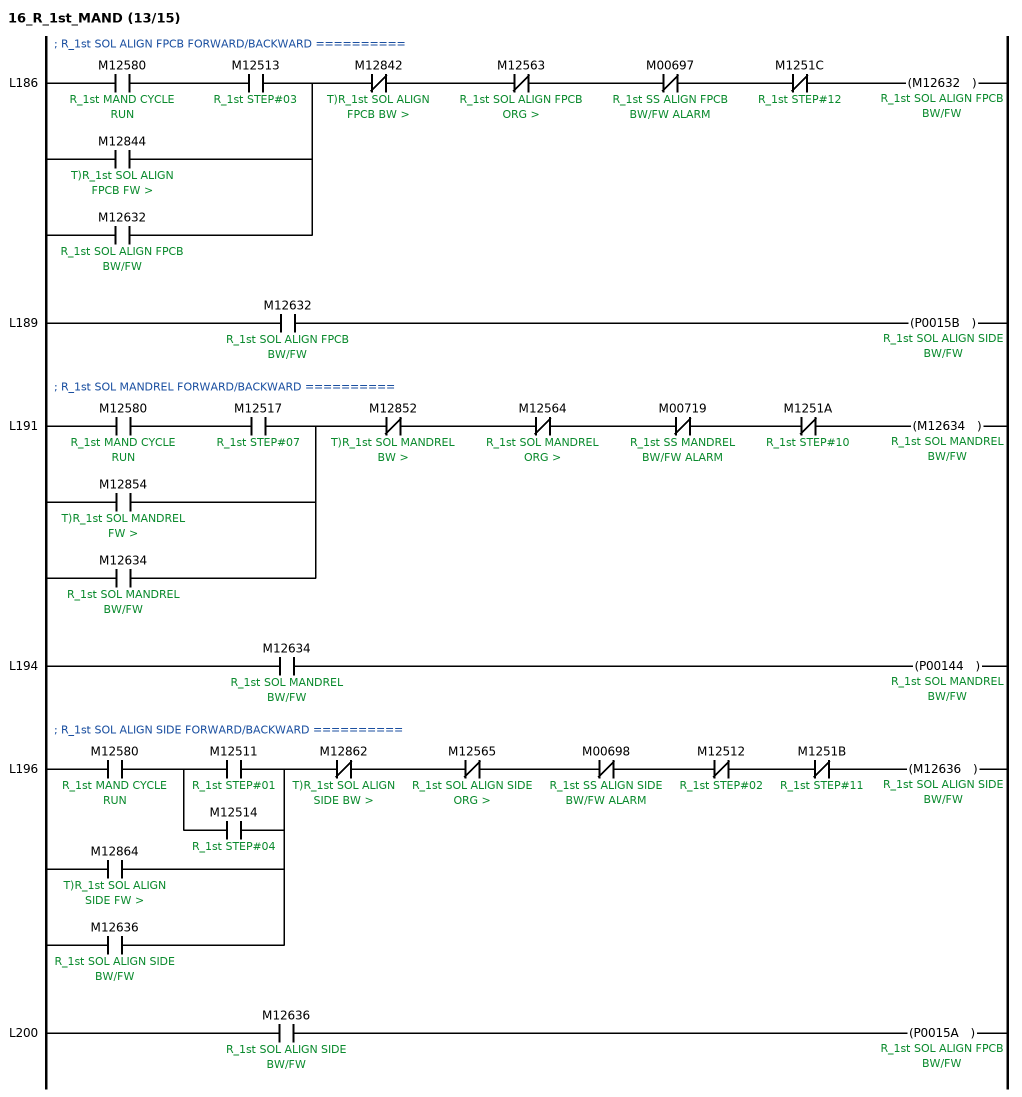
[picture p144: 16_R_1st_MAND rungs L186-L200]
// R_1st SOL ALIGN FPCB FORWARD/BACKWARD ==========
; L186
LOAD      M12580	// R_1st MAND CYCLE RUN
AND       M12513	// R_1st STEP#03
OR        M12844	// T)R_1st SOL ALIGN FPCB FW >
OR        M12632	// R_1st SOL ALIGN FPCB BW/FW
AND NOT   M12842	// T)R_1st SOL ALIGN FPCB BW >
AND NOT   M12563	// R_1st SOL ALIGN FPCB ORG >
AND NOT   M00697	// R_1st SS ALIGN FPCB BW/FW ALARM
AND NOT   M1251C	// R_1st STEP#12
OUT       M12632	// R_1st SOL ALIGN FPCB BW/FW
; L189
LOAD      M12632	// R_1st SOL ALIGN FPCB BW/FW
OUT       P0015B	// R_1st SOL ALIGN SIDE BW/FW
// R_1st SOL MANDREL FORWARD/BACKWARD ==========
; L191
LOAD      M12580	// R_1st MAND CYCLE RUN
AND       M12517	// R_1st STEP#07
OR        M12854	// T)R_1st SOL MANDREL FW >
OR        M12634	// R_1st SOL MANDREL BW/FW
AND NOT   M12852	// T)R_1st SOL MANDREL BW >
AND NOT   M12564	// R_1st SOL MANDREL ORG >
AND NOT   M00719	// R_1st SS MANDREL BW/FW ALARM
AND NOT   M1251A	// R_1st STEP#10
OUT       M12634	// R_1st SOL MANDREL BW/FW
; L194
LOAD      M12634	// R_1st SOL MANDREL BW/FW
OUT       P00144	// R_1st SOL MANDREL BW/FW
// R_1st SOL ALIGN SIDE FORWARD/BACKWARD ==========
; L196
LOAD      M12580	// R_1st MAND CYCLE RUN
LOAD      M12511	// R_1st STEP#01
OR        M12514	// R_1st STEP#04
AND LOAD
OR        M12864	// T)R_1st SOL ALIGN SIDE FW >
OR        M12636	// R_1st SOL ALIGN SIDE BW/FW
AND NOT   M12862	// T)R_1st SOL ALIGN SIDE BW >
AND NOT   M12565	// R_1st SOL ALIGN SIDE ORG >
AND NOT   M00698	// R_1st SS ALIGN SIDE BW/FW ALARM
AND NOT   M12512	// R_1st STEP#02
AND NOT   M1251B	// R_1st STEP#11
OUT       M12636	// R_1st SOL ALIGN SIDE BW/FW
; L200
LOAD      M12636	// R_1st SOL ALIGN SIDE BW/FW
OUT       P0015A	// R_1st SOL ALIGN FPCB BW/FW

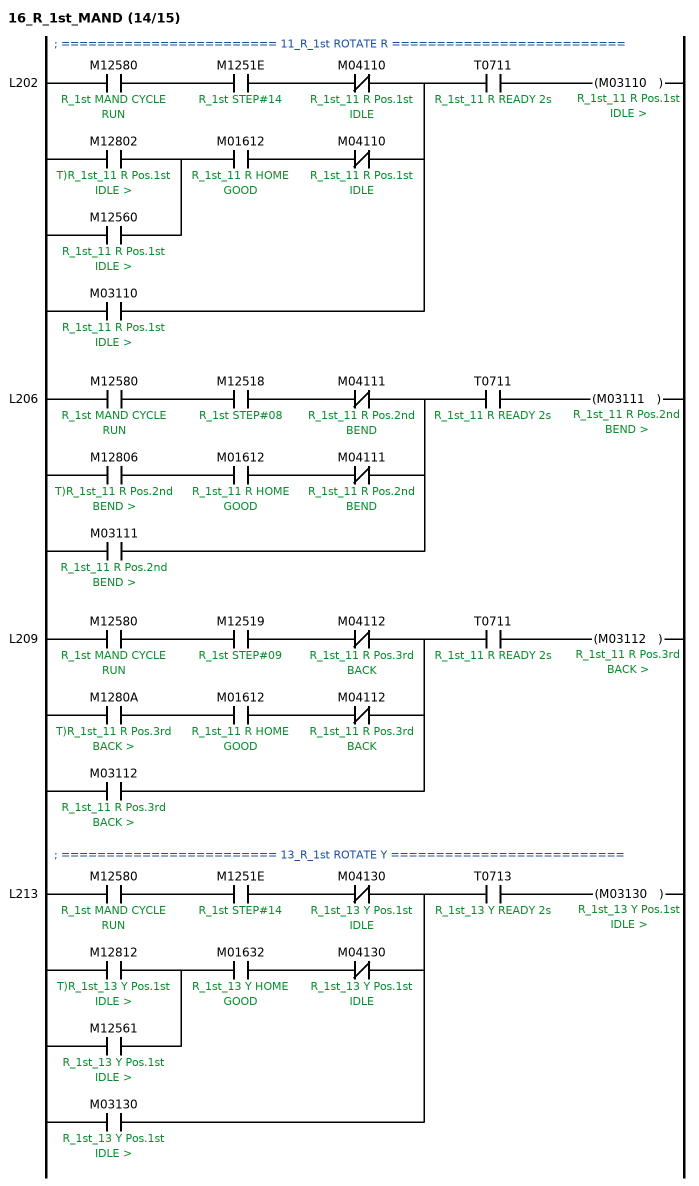
// ======================== 11_R_1st ROTATE R ==========================
; L202
LOAD      M12580	// R_1st MAND CYCLE RUN
AND       M1251E	// R_1st STEP#14
AND NOT   M04110	// R_1st_11 R Pos.1st IDLE
LOAD      M12802	// T)R_1st_11 R Pos.1st IDLE >
OR        M12560	// R_1st_11 R Pos.1st IDLE >
AND       M01612	// R_1st_11 R HOME GOOD
AND NOT   M04110	// R_1st_11 R Pos.1st IDLE
OR LOAD
OR        M03110	// R_1st_11 R Pos.1st IDLE >
AND       T0711	// R_1st_11 R READY 2s
OUT       M03110	// R_1st_11 R Pos.1st IDLE >
; L206
LOAD      M12580	// R_1st MAND CYCLE RUN
AND       M12518	// R_1st STEP#08
AND NOT   M04111	// R_1st_11 R Pos.2nd BEND
LOAD      M12806	// T)R_1st_11 R Pos.2nd BEND >
AND       M01612	// R_1st_11 R HOME GOOD
AND NOT   M04111	// R_1st_11 R Pos.2nd BEND
OR LOAD
OR        M03111	// R_1st_11 R Pos.2nd BEND >
AND       T0711	// R_1st_11 R READY 2s
OUT       M03111	// R_1st_11 R Pos.2nd BEND >
; L209
LOAD      M12580	// R_1st MAND CYCLE RUN
AND       M12519	// R_1st STEP#09
AND NOT   M04112	// R_1st_11 R Pos.3rd BACK
LOAD      M1280A	// T)R_1st_11 R Pos.3rd BACK >
AND       M01612	// R_1st_11 R HOME GOOD
AND NOT   M04112	// R_1st_11 R Pos.3rd BACK
OR LOAD
OR        M03112	// R_1st_11 R Pos.3rd BACK >
AND       T0711	// R_1st_11 R READY 2s
OUT       M03112	// R_1st_11 R Pos.3rd BACK >
// ======================== 13_R_1st ROTATE Y ==========================
; L213
LOAD      M12580	// R_1st MAND CYCLE RUN
AND       M1251E	// R_1st STEP#14
AND NOT   M04130	// R_1st_13 Y Pos.1st IDLE
LOAD      M12812	// T)R_1st_13 Y Pos.1st IDLE >
OR        M12561	// R_1st_13 Y Pos.1st IDLE >
AND       M01632	// R_1st_13 Y HOME GOOD
AND NOT   M04130	// R_1st_13 Y Pos.1st IDLE
OR LOAD
OR        M03130	// R_1st_13 Y Pos.1st IDLE >
AND       T0713	// R_1st_13 Y READY 2s
OUT       M03130	// R_1st_13 Y Pos.1st IDLE >

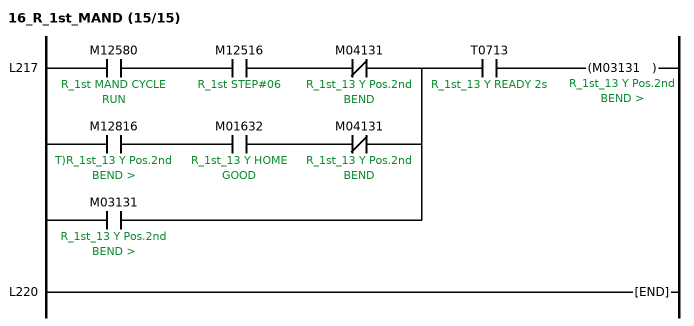
; L217
LOAD      M12580	// R_1st MAND CYCLE RUN
AND       M12516	// R_1st STEP#06
AND NOT   M04131	// R_1st_13 Y Pos.2nd BEND
LOAD      M12816	// T)R_1st_13 Y Pos.2nd BEND >
AND       M01632	// R_1st_13 Y HOME GOOD
AND NOT   M04131	// R_1st_13 Y Pos.2nd BEND
OR LOAD
OR        M03131	// R_1st_13 Y Pos.2nd BEND >
AND       T0713	// R_1st_13 Y READY 2s
OUT       M03131	// R_1st_13 Y Pos.2nd BEND >
; L220
END

PROGRAM 17_R_2nd_MAND (task: ¨ö¨¬A¥ì CA¡¤I¡¾¡¿¡¤¡Í)

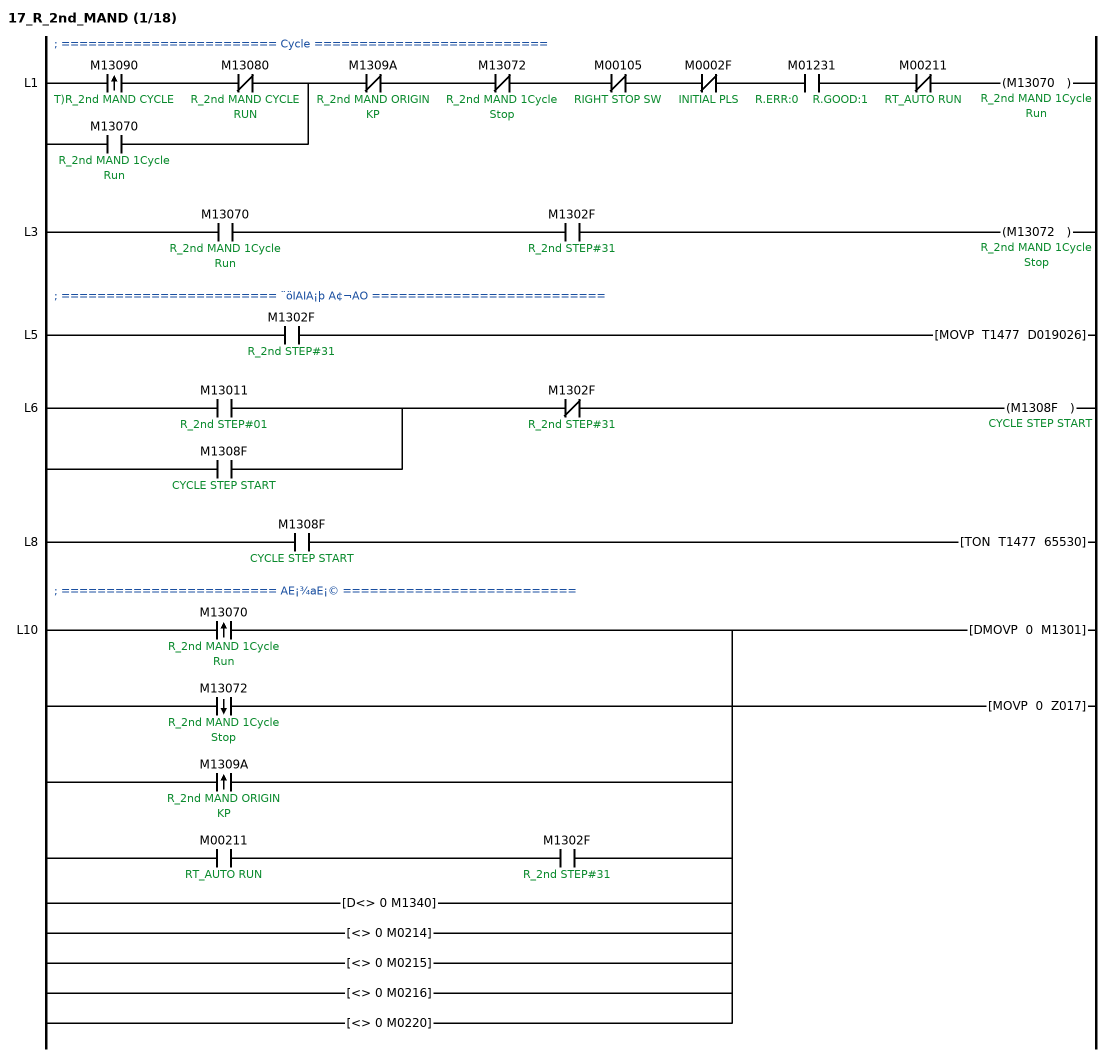
// ======================== Cycle ==========================
; L1
LOADP     M13090	// T)R_2nd MAND CYCLE
AND NOT   M13080	// R_2nd MAND CYCLE RUN
OR        M13070	// R_2nd MAND 1Cycle Run
AND NOT   M1309A	// R_2nd MAND ORIGIN KP
AND NOT   M13072	// R_2nd MAND 1Cycle Stop
AND NOT   M00105	// RIGHT STOP SW
AND NOT   M0002F	// INITIAL PLS
AND       M01231	// R.ERR:0    R.GOOD:1
AND NOT   M00211	// RT_AUTO RUN
OUT       M13070	// R_2nd MAND 1Cycle Run
; L3
LOAD      M13070	// R_2nd MAND 1Cycle Run
AND       M1302F	// R_2nd STEP#31
OUT       M13072	// R_2nd MAND 1Cycle Stop
// ======================== ¨öIAIA¡þ A¢¬AO ==========================
; L5
LOAD      M1302F	// R_2nd STEP#31
MOVP      T1477 D019026
; L6
LOAD      M13011	// R_2nd STEP#01
OR        M1308F	// CYCLE STEP START
AND NOT   M1302F	// R_2nd STEP#31
OUT       M1308F	// CYCLE STEP START
; L8
LOAD      M1308F	// CYCLE STEP START
TON       T1477 65530
// ======================== AE¡¾aE¡© ==========================
; L10
LOADP     M13070	// R_2nd MAND 1Cycle Run
ORN       M13072	// R_2nd MAND 1Cycle Stop
ORP       M1309A	// R_2nd MAND ORIGIN KP
LOAD      M00211	// RT_AUTO RUN
AND       M1302F	// R_2nd STEP#31
OR LOAD
ORD<>     0 M1340
OR<>      0 M0214
OR<>      0 M0215
OR<>      0 M0216
OR<>      0 M0220
DMOVP     0 M1301
MOVP      0 Z017

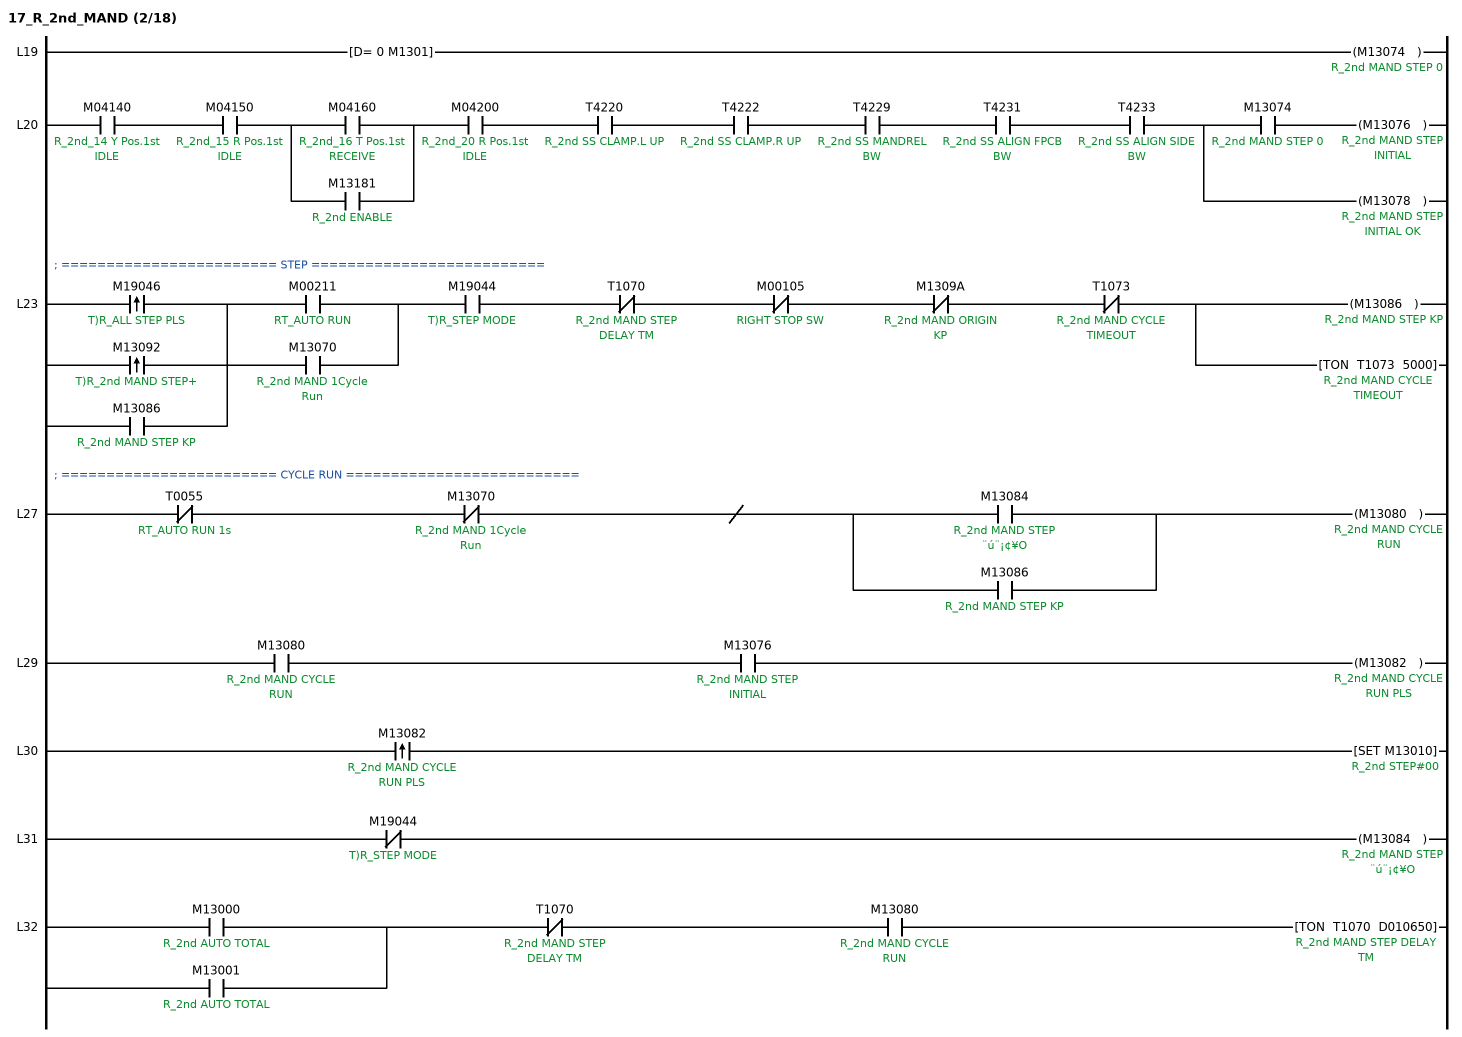
; L19
LOADD=    0 M1301
OUT       M13074	// R_2nd MAND STEP 0
; L20
LOAD      M04140	// R_2nd_14 Y Pos.1st IDLE
AND       M04150	// R_2nd_15 R Pos.1st IDLE
LOAD      M04160	// R_2nd_16 T Pos.1st RECEIVE
OR        M13181	// R_2nd ENABLE
AND LOAD
AND       M04200	// R_2nd_20 R Pos.1st IDLE
AND       T4220	// R_2nd SS CLAMP.L UP
AND       T4222	// R_2nd SS CLAMP.R UP
AND       T4229	// R_2nd SS MANDREL BW
AND       T4231	// R_2nd SS ALIGN FPCB BW
AND       T4233	// R_2nd SS ALIGN SIDE BW
MPUSH
AND       M13074	// R_2nd MAND STEP 0
OUT       M13076	// R_2nd MAND STEP INITIAL
MPOP
OUT       M13078	// R_2nd MAND STEP INITIAL OK
// ======================== STEP ==========================
; L23
LOADP     M19046	// T)R_ALL STEP PLS
ORP       M13092	// T)R_2nd MAND STEP+
OR        M13086	// R_2nd MAND STEP KP
LOAD      M00211	// RT_AUTO RUN
OR        M13070	// R_2nd MAND 1Cycle Run
AND LOAD
AND       M19044	// T)R_STEP MODE
AND NOT   T1070	// R_2nd MAND STEP DELAY TM
AND NOT   M00105	// RIGHT STOP SW
AND NOT   M1309A	// R_2nd MAND ORIGIN KP
AND NOT   T1073	// R_2nd MAND CYCLE TIMEOUT
OUT       M13086	// R_2nd MAND STEP KP
TON       T1073 5000	// R_2nd MAND CYCLE TIMEOUT
// ======================== CYCLE RUN ==========================
; L27
LOAD NOT  T0055	// RT_AUTO RUN 1s
AND NOT   M13070	// R_2nd MAND 1Cycle Run
NOT
LOAD      M13084	// R_2nd MAND STEP ¨ú¨¡¢¥O
OR        M13086	// R_2nd MAND STEP KP
AND LOAD
OUT       M13080	// R_2nd MAND CYCLE RUN
; L29
LOAD      M13080	// R_2nd MAND CYCLE RUN
AND       M13076	// R_2nd MAND STEP INITIAL
OUT       M13082	// R_2nd MAND CYCLE RUN PLS
; L30
LOADP     M13082	// R_2nd MAND CYCLE RUN PLS
SET       M13010	// R_2nd STEP#00
; L31
LOAD NOT  M19044	// T)R_STEP MODE
OUT       M13084	// R_2nd MAND STEP ¨ú¨¡¢¥O
; L32
LOAD      M13000	// R_2nd AUTO TOTAL
OR        M13001	// R_2nd AUTO TOTAL
AND NOT   T1070	// R_2nd MAND STEP DELAY TM
AND       M13080	// R_2nd MAND CYCLE RUN
TON       T1070 D010650	// R_2nd MAND STEP DELAY TM

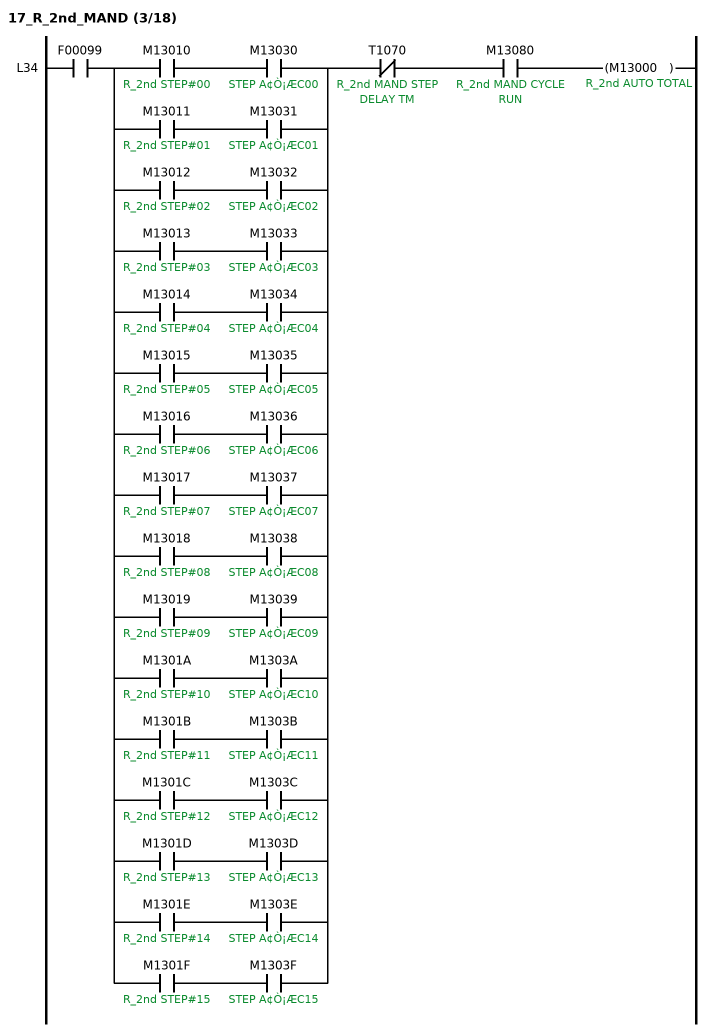
; L34
LOAD      F00099
LOAD      M13010	// R_2nd STEP#00
AND       M13030	// STEP A¢Ò¡ÆC00
LOAD      M13011	// R_2nd STEP#01
AND       M13031	// STEP A¢Ò¡ÆC01
OR LOAD
LOAD      M13012	// R_2nd STEP#02
AND       M13032	// STEP A¢Ò¡ÆC02
OR LOAD
LOAD      M13013	// R_2nd STEP#03
AND       M13033	// STEP A¢Ò¡ÆC03
OR LOAD
LOAD      M13014	// R_2nd STEP#04
AND       M13034	// STEP A¢Ò¡ÆC04
OR LOAD
LOAD      M13015	// R_2nd STEP#05
AND       M13035	// STEP A¢Ò¡ÆC05
OR LOAD
LOAD      M13016	// R_2nd STEP#06
AND       M13036	// STEP A¢Ò¡ÆC06
OR LOAD
LOAD      M13017	// R_2nd STEP#07
AND       M13037	// STEP A¢Ò¡ÆC07
OR LOAD
LOAD      M13018	// R_2nd STEP#08
AND       M13038	// STEP A¢Ò¡ÆC08
OR LOAD
LOAD      M13019	// R_2nd STEP#09
AND       M13039	// STEP A¢Ò¡ÆC09
OR LOAD
LOAD      M1301A	// R_2nd STEP#10
AND       M1303A	// STEP A¢Ò¡ÆC10
OR LOAD
LOAD      M1301B	// R_2nd STEP#11
AND       M1303B	// STEP A¢Ò¡ÆC11
OR LOAD
LOAD      M1301C	// R_2nd STEP#12
AND       M1303C	// STEP A¢Ò¡ÆC12
OR LOAD
LOAD      M1301D	// R_2nd STEP#13
AND       M1303D	// STEP A¢Ò¡ÆC13
OR LOAD
LOAD      M1301E	// R_2nd STEP#14
AND       M1303E	// STEP A¢Ò¡ÆC14
OR LOAD
LOAD      M1301F	// R_2nd STEP#15
AND       M1303F	// STEP A¢Ò¡ÆC15
OR LOAD
AND LOAD
AND NOT   T1070	// R_2nd MAND STEP DELAY TM
AND       M13080	// R_2nd MAND CYCLE RUN
OUT       M13000	// R_2nd AUTO TOTAL

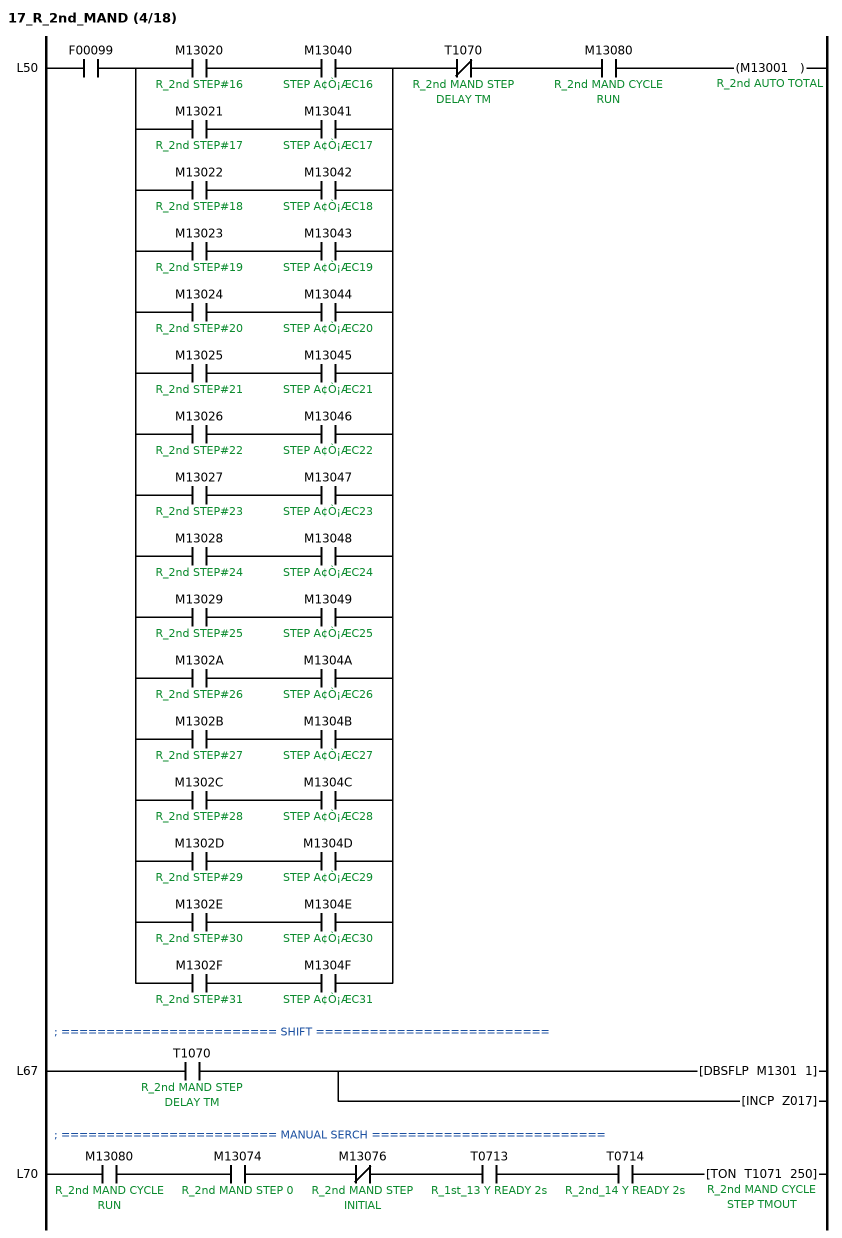
; L50
LOAD      F00099
LOAD      M13020	// R_2nd STEP#16
AND       M13040	// STEP A¢Ò¡ÆC16
LOAD      M13021	// R_2nd STEP#17
AND       M13041	// STEP A¢Ò¡ÆC17
OR LOAD
LOAD      M13022	// R_2nd STEP#18
AND       M13042	// STEP A¢Ò¡ÆC18
OR LOAD
LOAD      M13023	// R_2nd STEP#19
AND       M13043	// STEP A¢Ò¡ÆC19
OR LOAD
LOAD      M13024	// R_2nd STEP#20
AND       M13044	// STEP A¢Ò¡ÆC20
OR LOAD
LOAD      M13025	// R_2nd STEP#21
AND       M13045	// STEP A¢Ò¡ÆC21
OR LOAD
LOAD      M13026	// R_2nd STEP#22
AND       M13046	// STEP A¢Ò¡ÆC22
OR LOAD
LOAD      M13027	// R_2nd STEP#23
AND       M13047	// STEP A¢Ò¡ÆC23
OR LOAD
LOAD      M13028	// R_2nd STEP#24
AND       M13048	// STEP A¢Ò¡ÆC24
OR LOAD
LOAD      M13029	// R_2nd STEP#25
AND       M13049	// STEP A¢Ò¡ÆC25
OR LOAD
LOAD      M1302A	// R_2nd STEP#26
AND       M1304A	// STEP A¢Ò¡ÆC26
OR LOAD
LOAD      M1302B	// R_2nd STEP#27
AND       M1304B	// STEP A¢Ò¡ÆC27
OR LOAD
LOAD      M1302C	// R_2nd STEP#28
AND       M1304C	// STEP A¢Ò¡ÆC28
OR LOAD
LOAD      M1302D	// R_2nd STEP#29
AND       M1304D	// STEP A¢Ò¡ÆC29
OR LOAD
LOAD      M1302E	// R_2nd STEP#30
AND       M1304E	// STEP A¢Ò¡ÆC30
OR LOAD
LOAD      M1302F	// R_2nd STEP#31
AND       M1304F	// STEP A¢Ò¡ÆC31
OR LOAD
AND LOAD
AND NOT   T1070	// R_2nd MAND STEP DELAY TM
AND       M13080	// R_2nd MAND CYCLE RUN
OUT       M13001	// R_2nd AUTO TOTAL
// ======================== SHIFT ==========================
; L67
LOAD      T1070	// R_2nd MAND STEP DELAY TM
DBSFLP    M1301 1
INCP      Z017
// ======================== MANUAL SERCH ==========================
; L70
LOAD      M13080	// R_2nd MAND CYCLE RUN
AND       M13074	// R_2nd MAND STEP 0
AND NOT   M13076	// R_2nd MAND STEP INITIAL
AND       T0713	// R_1st_13 Y READY 2s
AND       T0714	// R_2nd_14 Y READY 2s
TON       T1071 250	// R_2nd MAND CYCLE STEP TMOUT

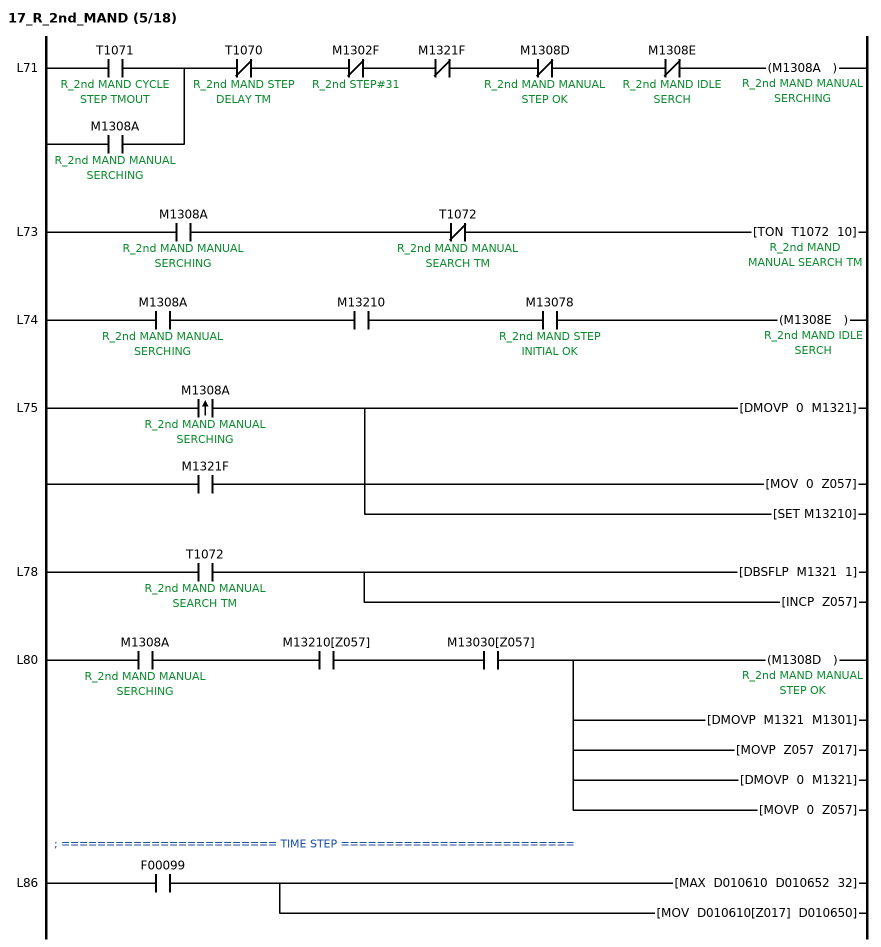
; L71
LOAD      T1071	// R_2nd MAND CYCLE STEP TMOUT
OR        M1308A	// R_2nd MAND MANUAL SERCHING
AND NOT   T1070	// R_2nd MAND STEP DELAY TM
AND NOT   M1302F	// R_2nd STEP#31
AND NOT   M1321F
AND NOT   M1308D	// R_2nd MAND MANUAL STEP OK
AND NOT   M1308E	// R_2nd MAND IDLE SERCH
OUT       M1308A	// R_2nd MAND MANUAL SERCHING
; L73
LOAD      M1308A	// R_2nd MAND MANUAL SERCHING
AND NOT   T1072	// R_2nd MAND MANUAL SEARCH TM
TON       T1072 10	// R_2nd MAND MANUAL SEARCH TM
; L74
LOAD      M1308A	// R_2nd MAND MANUAL SERCHING
AND       M13210
AND       M13078	// R_2nd MAND STEP INITIAL OK
OUT       M1308E	// R_2nd MAND IDLE SERCH
; L75
LOADP     M1308A	// R_2nd MAND MANUAL SERCHING
OR        M1321F
DMOVP     0 M1321
MOV       0 Z057
SET       M13210
; L78
LOAD      T1072	// R_2nd MAND MANUAL SEARCH TM
DBSFLP    M1321 1
INCP      Z057
; L80
LOAD      M1308A	// R_2nd MAND MANUAL SERCHING
AND       M13210[Z057]
AND       M13030[Z057]
OUT       M1308D	// R_2nd MAND MANUAL STEP OK
DMOVP     M1321 M1301
MOVP      Z057 Z017
DMOVP     0 M1321
MOVP      0 Z057
// ======================== TIME STEP ==========================
; L86
LOAD      F00099
MAX       D010610 D010652 32
MOV       D010610[Z017] D010650

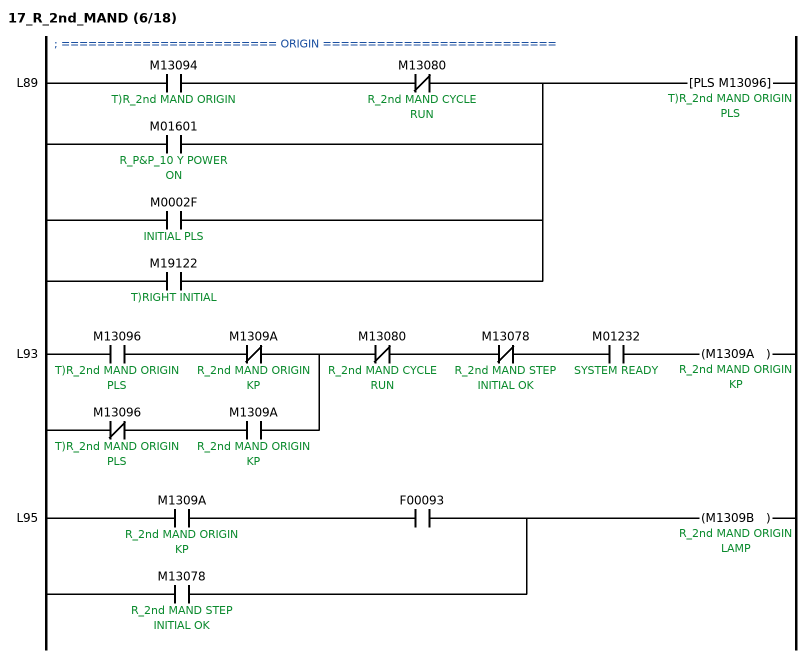
// ======================== ORIGIN ==========================
; L89
LOAD      M13094	// T)R_2nd MAND ORIGIN
AND NOT   M13080	// R_2nd MAND CYCLE RUN
OR        M01601	// R_P&P_10 Y POWER ON
OR        M0002F	// INITIAL PLS
OR        M19122	// T)RIGHT INITIAL
OUTP      M13096	// T)R_2nd MAND ORIGIN PLS
; L93
LOAD      M13096	// T)R_2nd MAND ORIGIN PLS
AND NOT   M1309A	// R_2nd MAND ORIGIN KP
LOAD NOT  M13096	// T)R_2nd MAND ORIGIN PLS
AND       M1309A	// R_2nd MAND ORIGIN KP
OR LOAD
AND NOT   M13080	// R_2nd MAND CYCLE RUN
AND NOT   M13078	// R_2nd MAND STEP INITIAL OK
AND       M01232	// SYSTEM READY
OUT       M1309A	// R_2nd MAND ORIGIN KP
; L95
LOAD      M1309A	// R_2nd MAND ORIGIN KP
AND       F00093
OR        M13078	// R_2nd MAND STEP INITIAL OK
OUT       M1309B	// R_2nd MAND ORIGIN LAMP

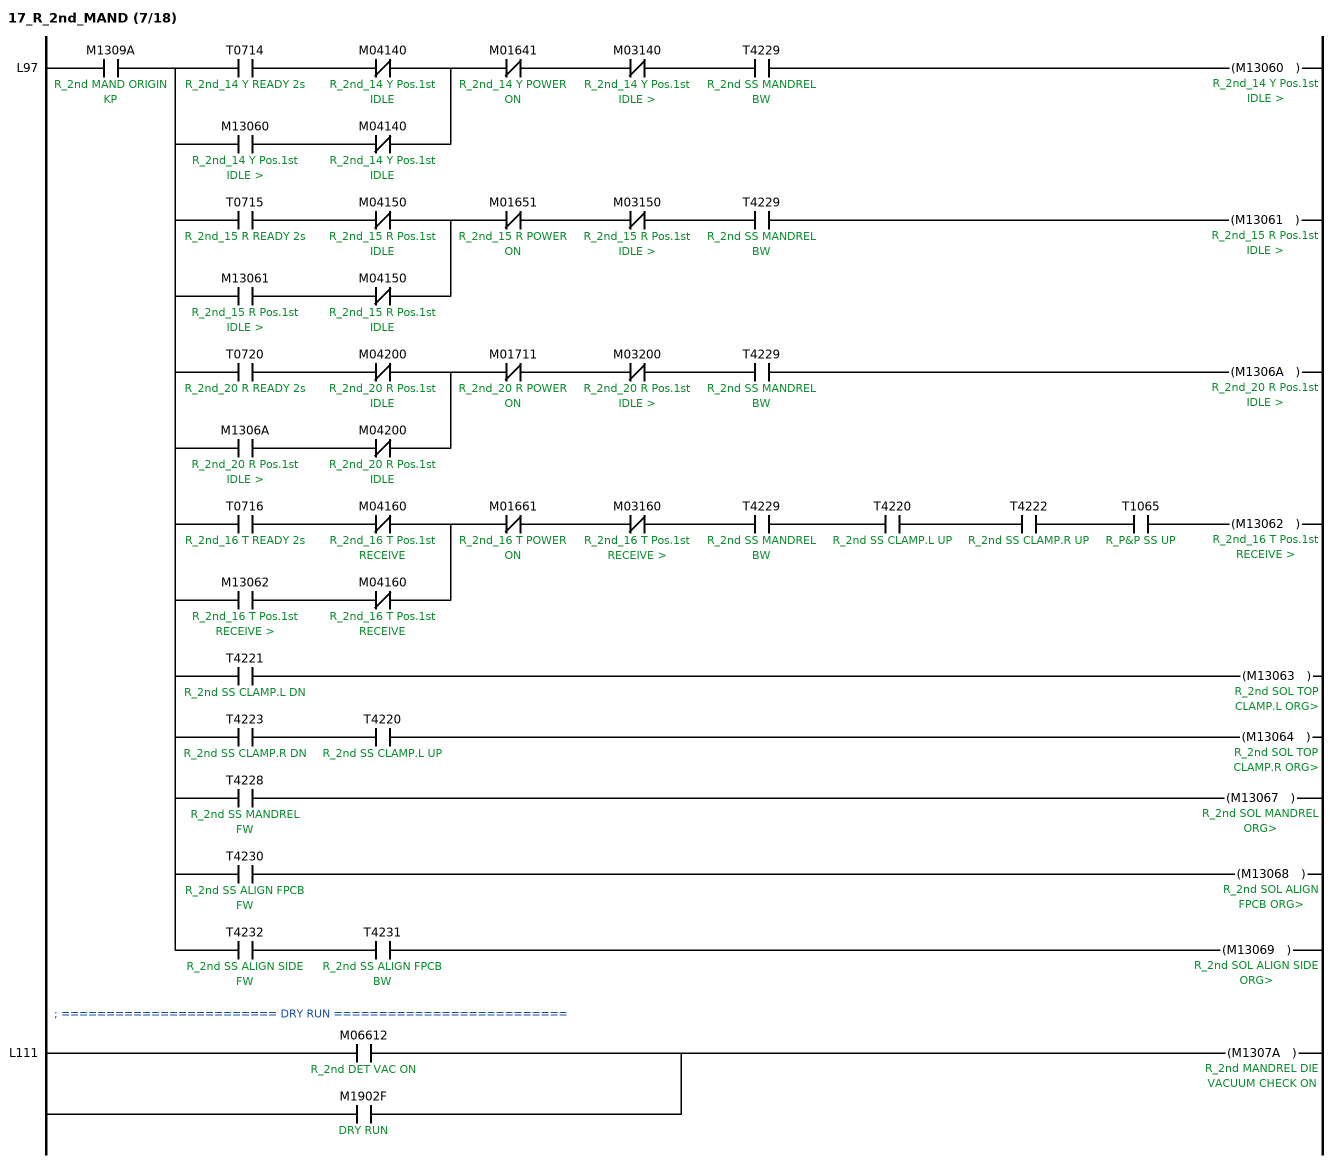
; L97
LOAD      M1309A	// R_2nd MAND ORIGIN KP
MPUSH
LOAD      T0714	// R_2nd_14 Y READY 2s
AND NOT   M04140	// R_2nd_14 Y Pos.1st IDLE
LOAD      M13060	// R_2nd_14 Y Pos.1st IDLE >
AND NOT   M04140	// R_2nd_14 Y Pos.1st IDLE
OR LOAD
AND LOAD
AND NOT   M01641	// R_2nd_14 Y POWER ON
AND NOT   M03140	// R_2nd_14 Y Pos.1st IDLE >
AND       T4229	// R_2nd SS MANDREL BW
OUT       M13060	// R_2nd_14 Y Pos.1st IDLE >
MLOAD
LOAD      T0715	// R_2nd_15 R READY 2s
AND NOT   M04150	// R_2nd_15 R Pos.1st IDLE
LOAD      M13061	// R_2nd_15 R Pos.1st IDLE >
AND NOT   M04150	// R_2nd_15 R Pos.1st IDLE
OR LOAD
AND LOAD
AND NOT   M01651	// R_2nd_15 R POWER ON
AND NOT   M03150	// R_2nd_15 R Pos.1st IDLE >
AND       T4229	// R_2nd SS MANDREL BW
OUT       M13061	// R_2nd_15 R Pos.1st IDLE >
MLOAD
LOAD      T0720	// R_2nd_20 R READY 2s
AND NOT   M04200	// R_2nd_20 R Pos.1st IDLE
LOAD      M1306A	// R_2nd_20 R Pos.1st IDLE >
AND NOT   M04200	// R_2nd_20 R Pos.1st IDLE
OR LOAD
AND LOAD
AND NOT   M01711	// R_2nd_20 R POWER ON
AND NOT   M03200	// R_2nd_20 R Pos.1st IDLE >
AND       T4229	// R_2nd SS MANDREL BW
OUT       M1306A	// R_2nd_20 R Pos.1st IDLE >
MLOAD
LOAD      T0716	// R_2nd_16 T READY 2s
AND NOT   M04160	// R_2nd_16 T Pos.1st RECEIVE
LOAD      M13062	// R_2nd_16 T Pos.1st RECEIVE >
AND NOT   M04160	// R_2nd_16 T Pos.1st RECEIVE
OR LOAD
AND LOAD
AND NOT   M01661	// R_2nd_16 T POWER ON
AND NOT   M03160	// R_2nd_16 T Pos.1st RECEIVE >
AND       T4229	// R_2nd SS MANDREL BW
AND       T4220	// R_2nd SS CLAMP.L UP
AND       T4222	// R_2nd SS CLAMP.R UP
AND       T1065	// R_P&P SS UP
OUT       M13062	// R_2nd_16 T Pos.1st RECEIVE >
MLOAD
AND       T4221	// R_2nd SS CLAMP.L DN
OUT       M13063	// R_2nd SOL TOP CLAMP.L ORG>
MLOAD
AND       T4223	// R_2nd SS CLAMP.R DN
AND       T4220	// R_2nd SS CLAMP.L UP
OUT       M13064	// R_2nd SOL TOP CLAMP.R ORG>
MLOAD
AND       T4228	// R_2nd SS MANDREL FW
OUT       M13067	// R_2nd SOL MANDREL ORG>
MLOAD
AND       T4230	// R_2nd SS ALIGN FPCB FW
OUT       M13068	// R_2nd SOL ALIGN FPCB ORG>
MPOP
AND       T4232	// R_2nd SS ALIGN SIDE FW
AND       T4231	// R_2nd SS ALIGN FPCB BW
OUT       M13069	// R_2nd SOL ALIGN SIDE ORG>
// ======================== DRY RUN ==========================
; L111
LOAD      M06612	// R_2nd DET VAC ON
OR        M1902F	// DRY RUN
OUT       M1307A	// R_2nd MANDREL DIE VACUUM CHECK ON

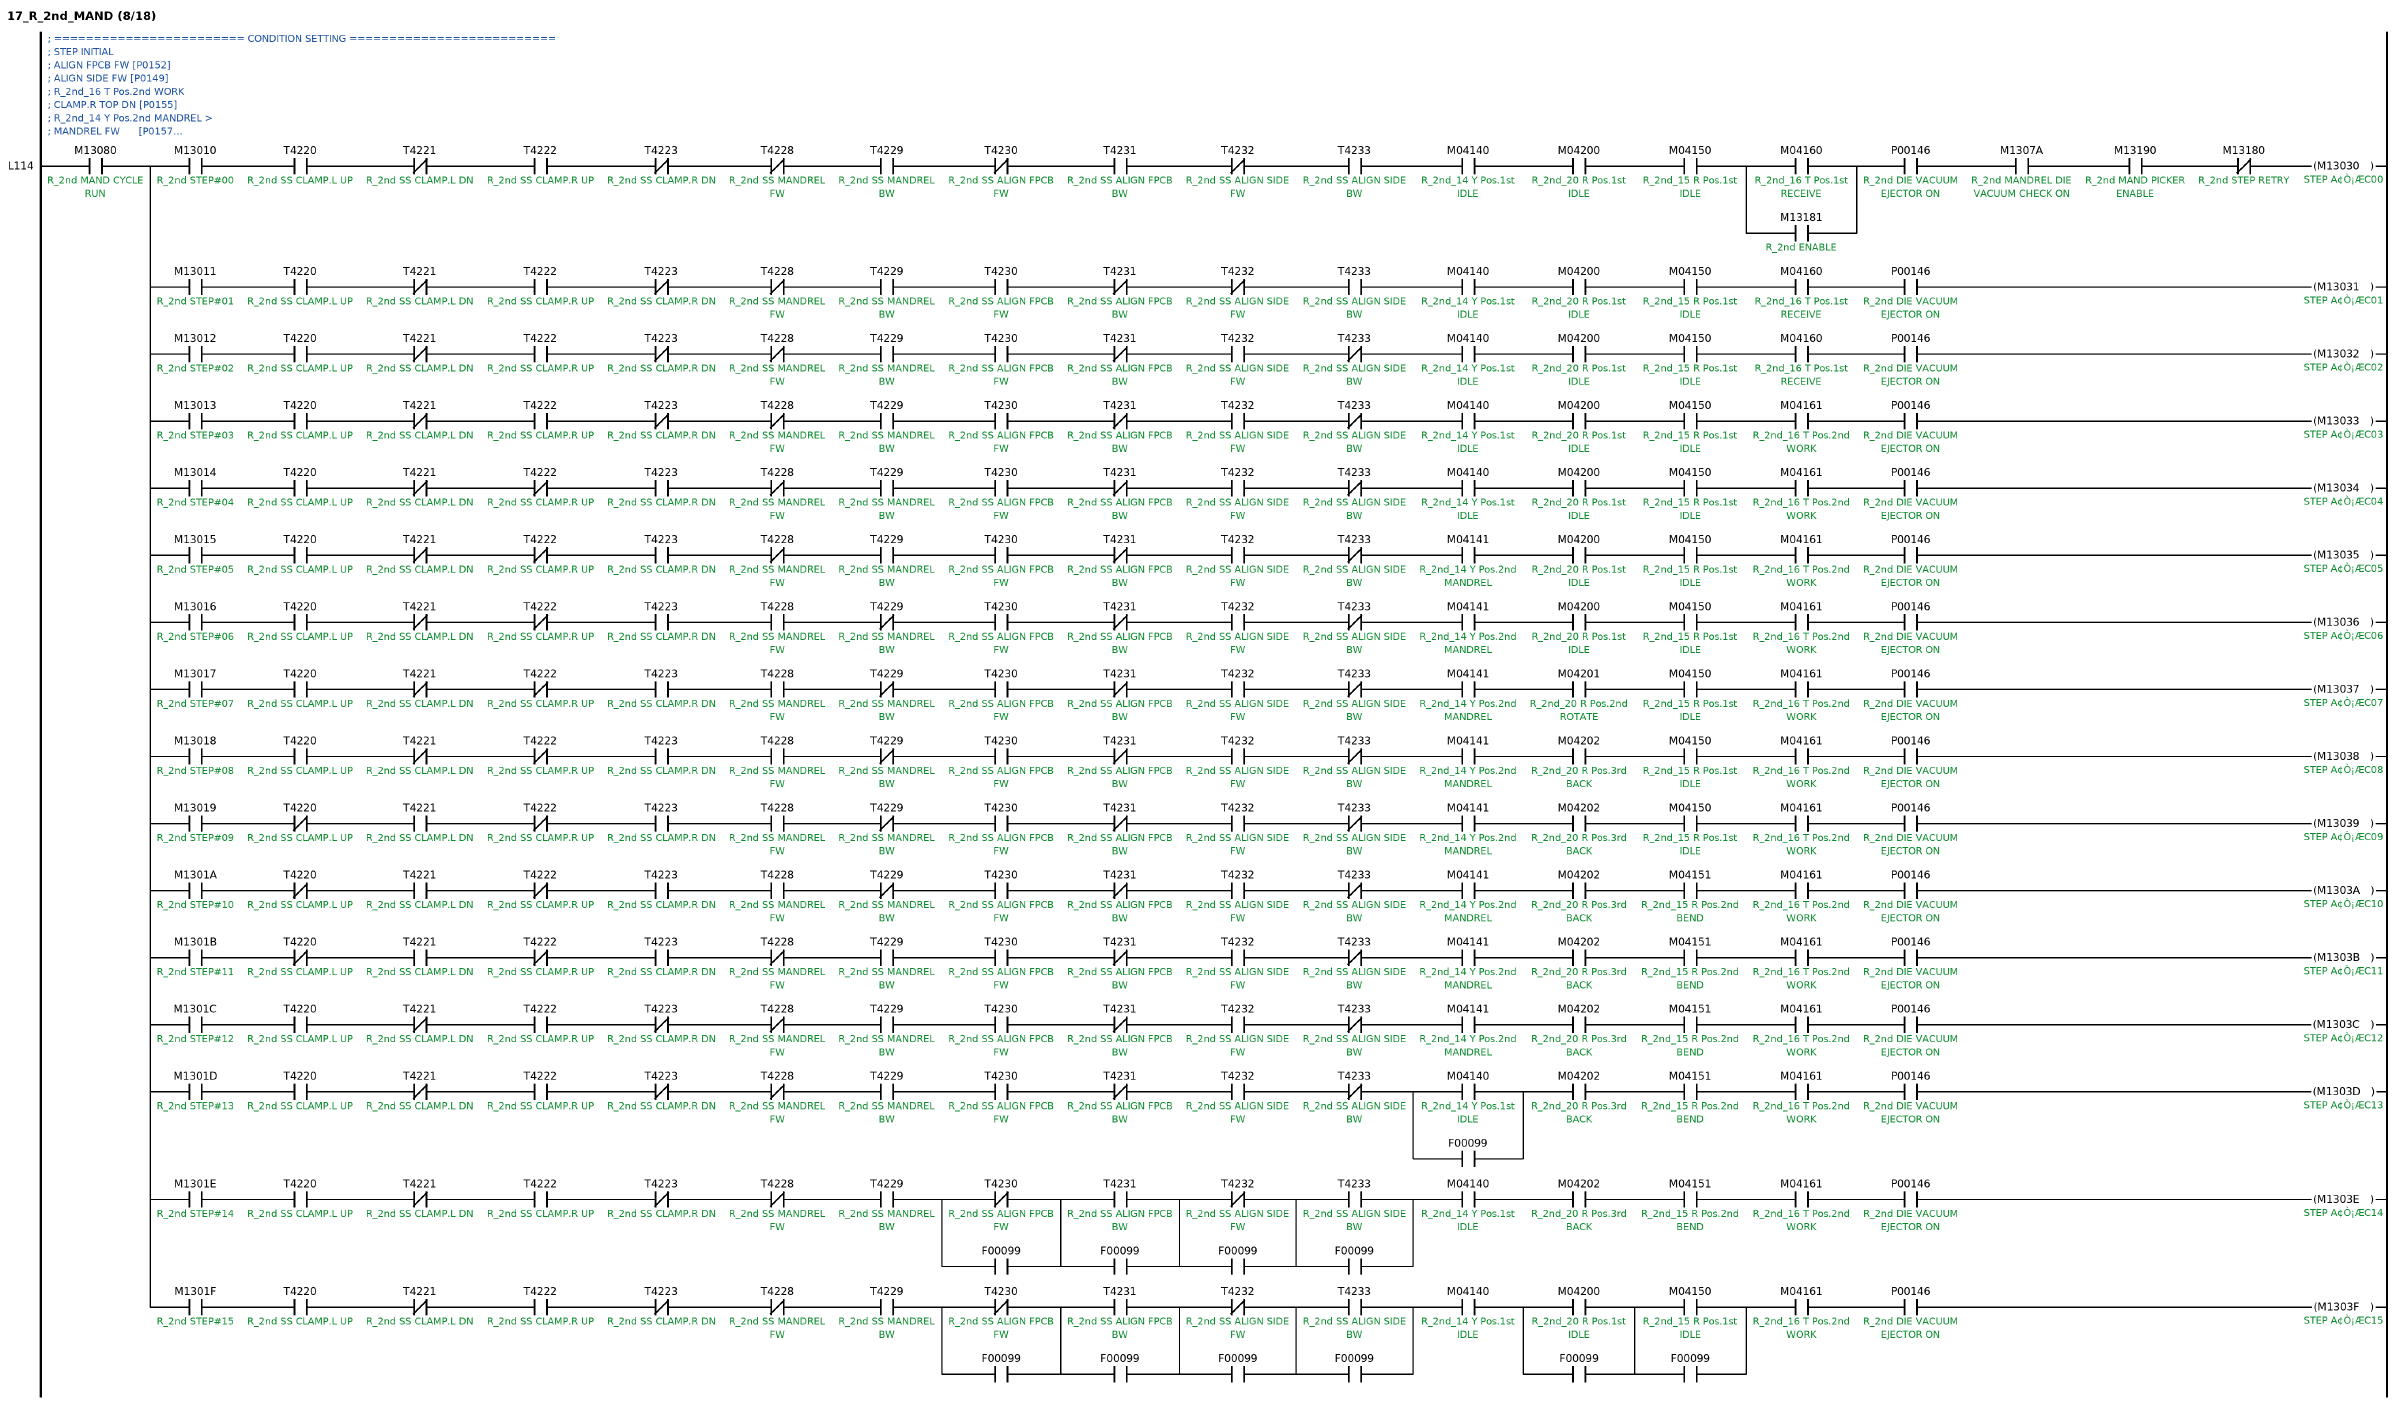
// ======================== CONDITION SETTING ==========================
; L114
LOAD      M13080	// R_2nd MAND CYCLE RUN
MPUSH
AND       M13010	// R_2nd STEP#00
AND       T4220	// R_2nd SS CLAMP.L UP
AND NOT   T4221	// R_2nd SS CLAMP.L DN
AND       T4222	// R_2nd SS CLAMP.R UP
AND NOT   T4223	// R_2nd SS CLAMP.R DN
AND NOT   T4228	// R_2nd SS MANDREL FW
AND       T4229	// R_2nd SS MANDREL BW
AND NOT   T4230	// R_2nd SS ALIGN FPCB FW
AND       T4231	// R_2nd SS ALIGN FPCB BW
AND NOT   T4232	// R_2nd SS ALIGN SIDE FW
AND       T4233	// R_2nd SS ALIGN SIDE BW
AND       M04140	// R_2nd_14 Y Pos.1st IDLE
AND       M04200	// R_2nd_20 R Pos.1st IDLE
AND       M04150	// R_2nd_15 R Pos.1st IDLE
LOAD      M04160	// R_2nd_16 T Pos.1st RECEIVE
OR        M13181	// R_2nd ENABLE
AND LOAD
AND       P00146	// R_2nd DIE VACUUM EJECTOR ON
AND       M1307A	// R_2nd MANDREL DIE VACUUM CHECK ON
AND       M13190	// R_2nd MAND PICKER ENABLE
AND NOT   M13180	// R_2nd STEP RETRY
OUT       M13030	// STEP A¢Ò¡ÆC00
MLOAD
AND       M13011	// R_2nd STEP#01
AND       T4220	// R_2nd SS CLAMP.L UP
AND NOT   T4221	// R_2nd SS CLAMP.L DN
AND       T4222	// R_2nd SS CLAMP.R UP
AND NOT   T4223	// R_2nd SS CLAMP.R DN
AND NOT   T4228	// R_2nd SS MANDREL FW
AND       T4229	// R_2nd SS MANDREL BW
AND       T4230	// R_2nd SS ALIGN FPCB FW
AND NOT   T4231	// R_2nd SS ALIGN FPCB BW
AND NOT   T4232	// R_2nd SS ALIGN SIDE FW
AND       T4233	// R_2nd SS ALIGN SIDE BW
AND       M04140	// R_2nd_14 Y Pos.1st IDLE
AND       M04200	// R_2nd_20 R Pos.1st IDLE
AND       M04150	// R_2nd_15 R Pos.1st IDLE
AND       M04160	// R_2nd_16 T Pos.1st RECEIVE
AND       P00146	// R_2nd DIE VACUUM EJECTOR ON
OUT       M13031	// STEP A¢Ò¡ÆC01
MLOAD
AND       M13012	// R_2nd STEP#02
AND       T4220	// R_2nd SS CLAMP.L UP
AND NOT   T4221	// R_2nd SS CLAMP.L DN
AND       T4222	// R_2nd SS CLAMP.R UP
AND NOT   T4223	// R_2nd SS CLAMP.R DN
AND NOT   T4228	// R_2nd SS MANDREL FW
AND       T4229	// R_2nd SS MANDREL BW
AND       T4230	// R_2nd SS ALIGN FPCB FW
AND NOT   T4231	// R_2nd SS ALIGN FPCB BW
AND       T4232	// R_2nd SS ALIGN SIDE FW
AND NOT   T4233	// R_2nd SS ALIGN SIDE BW
AND       M04140	// R_2nd_14 Y Pos.1st IDLE
AND       M04200	// R_2nd_20 R Pos.1st IDLE
AND       M04150	// R_2nd_15 R Pos.1st IDLE
AND       M04160	// R_2nd_16 T Pos.1st RECEIVE
AND       P00146	// R_2nd DIE VACUUM EJECTOR ON
OUT       M13032	// STEP A¢Ò¡ÆC02
MLOAD
AND       M13013	// R_2nd STEP#03
AND       T4220	// R_2nd SS CLAMP.L UP
AND NOT   T4221	// R_2nd SS CLAMP.L DN
AND       T4222	// R_2nd SS CLAMP.R UP
AND NOT   T4223	// R_2nd SS CLAMP.R DN
AND NOT   T4228	// R_2nd SS MANDREL FW
AND       T4229	// R_2nd SS MANDREL BW
AND       T4230	// R_2nd SS ALIGN FPCB FW
AND NOT   T4231	// R_2nd SS ALIGN FPCB BW
AND       T4232	// R_2nd SS ALIGN SIDE FW
AND NOT   T4233	// R_2nd SS ALIGN SIDE BW
AND       M04140	// R_2nd_14 Y Pos.1st IDLE
AND       M04200	// R_2nd_20 R Pos.1st IDLE
AND       M04150	// R_2nd_15 R Pos.1st IDLE
AND       M04161	// R_2nd_16 T Pos.2nd WORK
AND       P00146	// R_2nd DIE VACUUM EJECTOR ON
OUT       M13033	// STEP A¢Ò¡ÆC03
MLOAD
AND       M13014	// R_2nd STEP#04
AND       T4220	// R_2nd SS CLAMP.L UP
AND NOT   T4221	// R_2nd SS CLAMP.L DN
AND NOT   T4222	// R_2nd SS CLAMP.R UP
AND       T4223	// R_2nd SS CLAMP.R DN
AND NOT   T4228	// R_2nd SS MANDREL FW
AND       T4229	// R_2nd SS MANDREL BW
AND       T4230	// R_2nd SS ALIGN FPCB FW
AND NOT   T4231	// R_2nd SS ALIGN FPCB BW
AND       T4232	// R_2nd SS ALIGN SIDE FW
AND NOT   T4233	// R_2nd SS ALIGN SIDE BW
AND       M04140	// R_2nd_14 Y Pos.1st IDLE
AND       M04200	// R_2nd_20 R Pos.1st IDLE
AND       M04150	// R_2nd_15 R Pos.1st IDLE
AND       M04161	// R_2nd_16 T Pos.2nd WORK
AND       P00146	// R_2nd DIE VACUUM EJECTOR ON
OUT       M13034	// STEP A¢Ò¡ÆC04
MLOAD
AND       M13015	// R_2nd STEP#05
AND       T4220	// R_2nd SS CLAMP.L UP
AND NOT   T4221	// R_2nd SS CLAMP.L DN
AND NOT   T4222	// R_2nd SS CLAMP.R UP
AND       T4223	// R_2nd SS CLAMP.R DN
AND NOT   T4228	// R_2nd SS MANDREL FW
AND       T4229	// R_2nd SS MANDREL BW
AND       T4230	// R_2nd SS ALIGN FPCB FW
AND NOT   T4231	// R_2nd SS ALIGN FPCB BW
AND       T4232	// R_2nd SS ALIGN SIDE FW
AND NOT   T4233	// R_2nd SS ALIGN SIDE BW
AND       M04141	// R_2nd_14 Y Pos.2nd MANDREL
AND       M04200	// R_2nd_20 R Pos.1st IDLE
AND       M04150	// R_2nd_15 R Pos.1st IDLE
AND       M04161	// R_2nd_16 T Pos.2nd WORK
AND       P00146	// R_2nd DIE VACUUM EJECTOR ON
OUT       M13035	// STEP A¢Ò¡ÆC05
MLOAD
AND       M13016	// R_2nd STEP#06
AND       T4220	// R_2nd SS CLAMP.L UP
AND NOT   T4221	// R_2nd SS CLAMP.L DN
AND NOT   T4222	// R_2nd SS CLAMP.R UP
AND       T4223	// R_2nd SS CLAMP.R DN
AND       T4228	// R_2nd SS MANDREL FW
AND NOT   T4229	// R_2nd SS MANDREL BW
AND       T4230	// R_2nd SS ALIGN FPCB FW
AND NOT   T4231	// R_2nd SS ALIGN FPCB BW
AND       T4232	// R_2nd SS ALIGN SIDE FW
AND NOT   T4233	// R_2nd SS ALIGN SIDE BW
AND       M04141	// R_2nd_14 Y Pos.2nd MANDREL
AND       M04200	// R_2nd_20 R Pos.1st IDLE
AND       M04150	// R_2nd_15 R Pos.1st IDLE
AND       M04161	// R_2nd_16 T Pos.2nd WORK
AND       P00146	// R_2nd DIE VACUUM EJECTOR ON
OUT       M13036	// STEP A¢Ò¡ÆC06
MLOAD
AND       M13017	// R_2nd STEP#07
AND       T4220	// R_2nd SS CLAMP.L UP
AND NOT   T4221	// R_2nd SS CLAMP.L DN
AND NOT   T4222	// R_2nd SS CLAMP.R UP
AND       T4223	// R_2nd SS CLAMP.R DN
AND       T4228	// R_2nd SS MANDREL FW
AND NOT   T4229	// R_2nd SS MANDREL BW
AND       T4230	// R_2nd SS ALIGN FPCB FW
AND NOT   T4231	// R_2nd SS ALIGN FPCB BW
AND       T4232	// R_2nd SS ALIGN SIDE FW
AND NOT   T4233	// R_2nd SS ALIGN SIDE BW
AND       M04141	// R_2nd_14 Y Pos.2nd MANDREL
AND       M04201	// R_2nd_20 R Pos.2nd ROTATE
AND       M04150	// R_2nd_15 R Pos.1st IDLE
AND       M04161	// R_2nd_16 T Pos.2nd WORK
AND       P00146	// R_2nd DIE VACUUM EJECTOR ON
OUT       M13037	// STEP A¢Ò¡ÆC07
MLOAD
AND       M13018	// R_2nd STEP#08
AND       T4220	// R_2nd SS CLAMP.L UP
AND NOT   T4221	// R_2nd SS CLAMP.L DN
AND NOT   T4222	// R_2nd SS CLAMP.R UP
AND       T4223	// R_2nd SS CLAMP.R DN
AND       T4228	// R_2nd SS MANDREL FW
AND NOT   T4229	// R_2nd SS MANDREL BW
AND       T4230	// R_2nd SS ALIGN FPCB FW
AND NOT   T4231	// R_2nd SS ALIGN FPCB BW
AND       T4232	// R_2nd SS ALIGN SIDE FW
AND NOT   T4233	// R_2nd SS ALIGN SIDE BW
AND       M04141	// R_2nd_14 Y Pos.2nd MANDREL
AND       M04202	// R_2nd_20 R Pos.3rd BACK
AND       M04150	// R_2nd_15 R Pos.1st IDLE
AND       M04161	// R_2nd_16 T Pos.2nd WORK
AND       P00146	// R_2nd DIE VACUUM EJECTOR ON
OUT       M13038	// STEP A¢Ò¡ÆC08
MLOAD
AND       M13019	// R_2nd STEP#09
AND NOT   T4220	// R_2nd SS CLAMP.L UP
AND       T4221	// R_2nd SS CLAMP.L DN
AND NOT   T4222	// R_2nd SS CLAMP.R UP
AND       T4223	// R_2nd SS CLAMP.R DN
AND       T4228	// R_2nd SS MANDREL FW
AND NOT   T4229	// R_2nd SS MANDREL BW
AND       T4230	// R_2nd SS ALIGN FPCB FW
AND NOT   T4231	// R_2nd SS ALIGN FPCB BW
AND       T4232	// R_2nd SS ALIGN SIDE FW
AND NOT   T4233	// R_2nd SS ALIGN SIDE BW
AND       M04141	// R_2nd_14 Y Pos.2nd MANDREL
AND       M04202	// R_2nd_20 R Pos.3rd BACK
AND       M04150	// R_2nd_15 R Pos.1st IDLE
AND       M04161	// R_2nd_16 T Pos.2nd WORK
AND       P00146	// R_2nd DIE VACUUM EJECTOR ON
OUT       M13039	// STEP A¢Ò¡ÆC09
MLOAD
AND       M1301A	// R_2nd STEP#10
AND NOT   T4220	// R_2nd SS CLAMP.L UP
AND       T4221	// R_2nd SS CLAMP.L DN
AND NOT   T4222	// R_2nd SS CLAMP.R UP
AND       T4223	// R_2nd SS CLAMP.R DN
AND       T4228	// R_2nd SS MANDREL FW
AND NOT   T4229	// R_2nd SS MANDREL BW
AND       T4230	// R_2nd SS ALIGN FPCB FW
AND NOT   T4231	// R_2nd SS ALIGN FPCB BW
AND       T4232	// R_2nd SS ALIGN SIDE FW
AND NOT   T4233	// R_2nd SS ALIGN SIDE BW
AND       M04141	// R_2nd_14 Y Pos.2nd MANDREL
AND       M04202	// R_2nd_20 R Pos.3rd BACK
AND       M04151	// R_2nd_15 R Pos.2nd BEND
AND       M04161	// R_2nd_16 T Pos.2nd WORK
AND       P00146	// R_2nd DIE VACUUM EJECTOR ON
OUT       M1303A	// STEP A¢Ò¡ÆC10
MLOAD
AND       M1301B	// R_2nd STEP#11
AND NOT   T4220	// R_2nd SS CLAMP.L UP
AND       T4221	// R_2nd SS CLAMP.L DN
AND NOT   T4222	// R_2nd SS CLAMP.R UP
AND       T4223	// R_2nd SS CLAMP.R DN
AND NOT   T4228	// R_2nd SS MANDREL FW
AND       T4229	// R_2nd SS MANDREL BW
AND       T4230	// R_2nd SS ALIGN FPCB FW
AND NOT   T4231	// R_2nd SS ALIGN FPCB BW
AND       T4232	// R_2nd SS ALIGN SIDE FW
AND NOT   T4233	// R_2nd SS ALIGN SIDE BW
AND       M04141	// R_2nd_14 Y Pos.2nd MANDREL
AND       M04202	// R_2nd_20 R Pos.3rd BACK
AND       M04151	// R_2nd_15 R Pos.2nd BEND
AND       M04161	// R_2nd_16 T Pos.2nd WORK
AND       P00146	// R_2nd DIE VACUUM EJECTOR ON
OUT       M1303B	// STEP A¢Ò¡ÆC11
MLOAD
AND       M1301C	// R_2nd STEP#12
AND       T4220	// R_2nd SS CLAMP.L UP
AND NOT   T4221	// R_2nd SS CLAMP.L DN
AND       T4222	// R_2nd SS CLAMP.R UP
AND NOT   T4223	// R_2nd SS CLAMP.R DN
AND NOT   T4228	// R_2nd SS MANDREL FW
AND       T4229	// R_2nd SS MANDREL BW
AND       T4230	// R_2nd SS ALIGN FPCB FW
AND NOT   T4231	// R_2nd SS ALIGN FPCB BW
AND       T4232	// R_2nd SS ALIGN SIDE FW
AND NOT   T4233	// R_2nd SS ALIGN SIDE BW
AND       M04141	// R_2nd_14 Y Pos.2nd MANDREL
AND       M04202	// R_2nd_20 R Pos.3rd BACK
AND       M04151	// R_2nd_15 R Pos.2nd BEND
AND       M04161	// R_2nd_16 T Pos.2nd WORK
AND       P00146	// R_2nd DIE VACUUM EJECTOR ON
OUT       M1303C	// STEP A¢Ò¡ÆC12
MLOAD
AND       M1301D	// R_2nd STEP#13
AND       T4220	// R_2nd SS CLAMP.L UP
AND NOT   T4221	// R_2nd SS CLAMP.L DN
AND       T4222	// R_2nd SS CLAMP.R UP
AND NOT   T4223	// R_2nd SS CLAMP.R DN
AND NOT   T4228	// R_2nd SS MANDREL FW
AND       T4229	// R_2nd SS MANDREL BW
AND       T4230	// R_2nd SS ALIGN FPCB FW
AND NOT   T4231	// R_2nd SS ALIGN FPCB BW
AND       T4232	// R_2nd SS ALIGN SIDE FW
AND NOT   T4233	// R_2nd SS ALIGN SIDE BW
LOAD      M04140	// R_2nd_14 Y Pos.1st IDLE
OR        F00099
AND LOAD
AND       M04202	// R_2nd_20 R Pos.3rd BACK
AND       M04151	// R_2nd_15 R Pos.2nd BEND
AND       M04161	// R_2nd_16 T Pos.2nd WORK
AND       P00146	// R_2nd DIE VACUUM EJECTOR ON
OUT       M1303D	// STEP A¢Ò¡ÆC13
MLOAD
AND       M1301E	// R_2nd STEP#14
AND       T4220	// R_2nd SS CLAMP.L UP
AND NOT   T4221	// R_2nd SS CLAMP.L DN
AND       T4222	// R_2nd SS CLAMP.R UP
AND NOT   T4223	// R_2nd SS CLAMP.R DN
AND NOT   T4228	// R_2nd SS MANDREL FW
AND       T4229	// R_2nd SS MANDREL BW
LOAD NOT  T4230	// R_2nd SS ALIGN FPCB FW
OR        F00099
AND LOAD
LOAD      T4231	// R_2nd SS ALIGN FPCB BW
OR        F00099
AND LOAD
LOAD NOT  T4232	// R_2nd SS ALIGN SIDE FW
OR        F00099
AND LOAD
LOAD      T4233	// R_2nd SS ALIGN SIDE BW
OR        F00099
AND LOAD
AND       M04140	// R_2nd_14 Y Pos.1st IDLE
AND       M04202	// R_2nd_20 R Pos.3rd BACK
AND       M04151	// R_2nd_15 R Pos.2nd BEND
AND       M04161	// R_2nd_16 T Pos.2nd WORK
AND       P00146	// R_2nd DIE VACUUM EJECTOR ON
OUT       M1303E	// STEP A¢Ò¡ÆC14
MPOP
AND       M1301F	// R_2nd STEP#15
AND       T4220	// R_2nd SS CLAMP.L UP
AND NOT   T4221	// R_2nd SS CLAMP.L DN
AND       T4222	// R_2nd SS CLAMP.R UP
AND NOT   T4223	// R_2nd SS CLAMP.R DN
AND NOT   T4228	// R_2nd SS MANDREL FW
AND       T4229	// R_2nd SS MANDREL BW
LOAD NOT  T4230	// R_2nd SS ALIGN FPCB FW
OR        F00099
AND LOAD
LOAD      T4231	// R_2nd SS ALIGN FPCB BW
OR        F00099
AND LOAD
LOAD NOT  T4232	// R_2nd SS ALIGN SIDE FW
OR        F00099
AND LOAD
LOAD      T4233	// R_2nd SS ALIGN SIDE BW
OR        F00099
AND LOAD
AND       M04140	// R_2nd_14 Y Pos.1st IDLE
LOAD      M04200	// R_2nd_20 R Pos.1st IDLE
OR        F00099
AND LOAD
LOAD      M04150	// R_2nd_15 R Pos.1st IDLE
OR        F00099
AND LOAD
AND       M04161	// R_2nd_16 T Pos.2nd WORK
AND       P00146	// R_2nd DIE VACUUM EJECTOR ON
OUT       M1303F	// STEP A¢Ò¡ÆC15
// output comment: STEP INITIAL
// output comment: ALIGN FPCB FW [P0152]
// output comment: ALIGN SIDE FW [P0149]
// output comment: R_2nd_16 T Pos.2nd WORK
// output comment: CLAMP.R TOP DN [P0155]
// output comment: R_2nd_14 Y Pos.2nd MANDREL >
// output comment: MANDREL FW      [P0157]
// output comment: R_2nd_20 R Pos.2nd BEND >
// output comment: R_2nd_20 R Pos.3rd BACK >
// output comment: CLAMP.L TOP DN [P0156]
// output comment: R_2nd_15 R Pos.2nd ROTATE >
// output comment: MANDREL BW      [P0157]
// output comment: CLAMP TOP UP   [P0155-P0156]
// output comment: R_2nd_14 Y Pos.1st IDLE >
// output comment: ALIGN FPCB BW [P0152]                      ALIGN SIDE BW           [P0153]
// output comment: R_2nd_15 R Pos.1st IDLE >                    R_2nd_20 R Pos.1st IDLE >

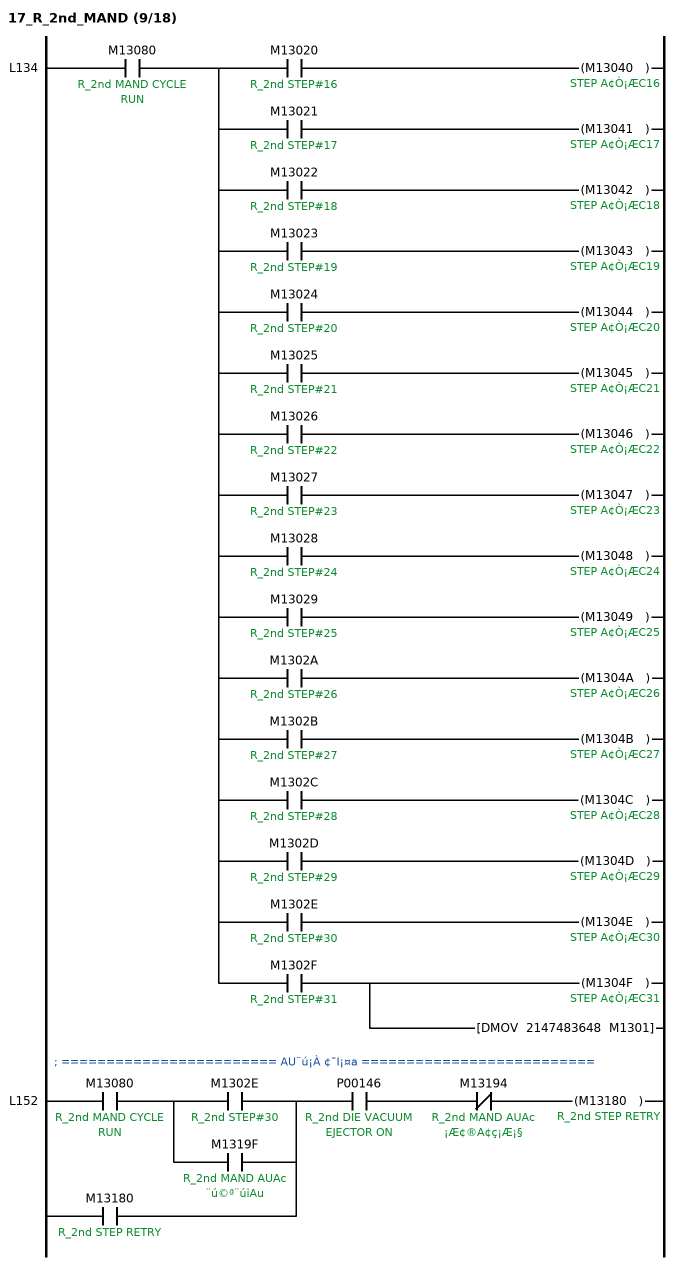
; L134
LOAD      M13080	// R_2nd MAND CYCLE RUN
MPUSH
AND       M13020	// R_2nd STEP#16
OUT       M13040	// STEP A¢Ò¡ÆC16
MLOAD
AND       M13021	// R_2nd STEP#17
OUT       M13041	// STEP A¢Ò¡ÆC17
MLOAD
AND       M13022	// R_2nd STEP#18
OUT       M13042	// STEP A¢Ò¡ÆC18
MLOAD
AND       M13023	// R_2nd STEP#19
OUT       M13043	// STEP A¢Ò¡ÆC19
MLOAD
AND       M13024	// R_2nd STEP#20
OUT       M13044	// STEP A¢Ò¡ÆC20
MLOAD
AND       M13025	// R_2nd STEP#21
OUT       M13045	// STEP A¢Ò¡ÆC21
MLOAD
AND       M13026	// R_2nd STEP#22
OUT       M13046	// STEP A¢Ò¡ÆC22
MLOAD
AND       M13027	// R_2nd STEP#23
OUT       M13047	// STEP A¢Ò¡ÆC23
MLOAD
AND       M13028	// R_2nd STEP#24
OUT       M13048	// STEP A¢Ò¡ÆC24
MLOAD
AND       M13029	// R_2nd STEP#25
OUT       M13049	// STEP A¢Ò¡ÆC25
MLOAD
AND       M1302A	// R_2nd STEP#26
OUT       M1304A	// STEP A¢Ò¡ÆC26
MLOAD
AND       M1302B	// R_2nd STEP#27
OUT       M1304B	// STEP A¢Ò¡ÆC27
MLOAD
AND       M1302C	// R_2nd STEP#28
OUT       M1304C	// STEP A¢Ò¡ÆC28
MLOAD
AND       M1302D	// R_2nd STEP#29
OUT       M1304D	// STEP A¢Ò¡ÆC29
MLOAD
AND       M1302E	// R_2nd STEP#30
OUT       M1304E	// STEP A¢Ò¡ÆC30
MPOP
AND       M1302F	// R_2nd STEP#31
OUT       M1304F	// STEP A¢Ò¡ÆC31
DMOV      2147483648 M1301
// ======================== AU¨ú¡À ¢¯I¡¤a ==========================
; L152
LOAD      M13080	// R_2nd MAND CYCLE RUN
LOAD      M1302E	// R_2nd STEP#30
OR        M1319F	// R_2nd MAND AUAc ¨ú©ª¨úiAu
AND LOAD
OR        M13180	// R_2nd STEP RETRY
AND       P00146	// R_2nd DIE VACUUM EJECTOR ON
AND NOT   M13194	// R_2nd MAND AUAc ¡Æ¢®A¢ç¡Æ¡§
OUT       M13180	// R_2nd STEP RETRY

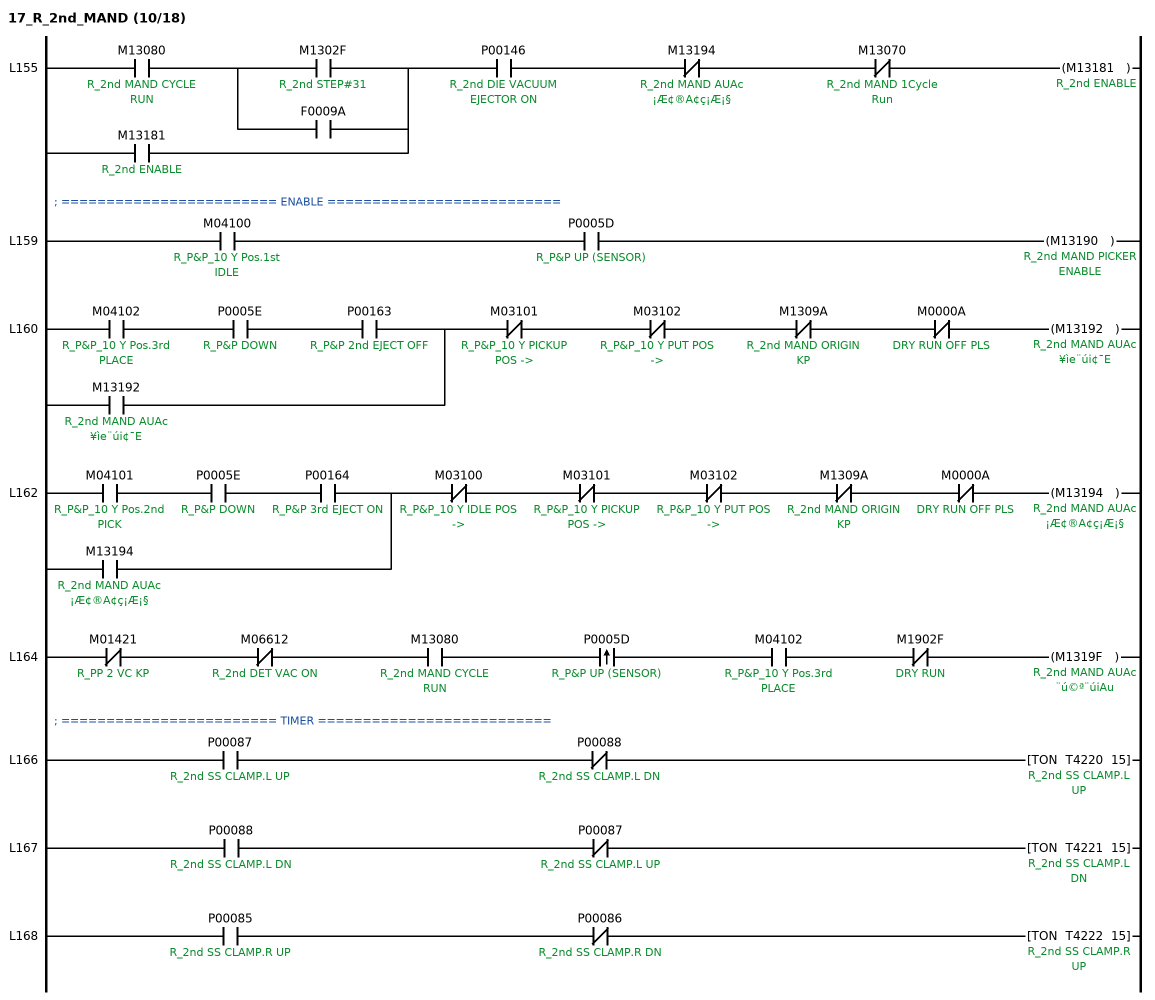
; L155
LOAD      M13080	// R_2nd MAND CYCLE RUN
LOAD      M1302F	// R_2nd STEP#31
OR        F0009A
AND LOAD
OR        M13181	// R_2nd ENABLE
AND       P00146	// R_2nd DIE VACUUM EJECTOR ON
AND NOT   M13194	// R_2nd MAND AUAc ¡Æ¢®A¢ç¡Æ¡§
AND NOT   M13070	// R_2nd MAND 1Cycle Run
OUT       M13181	// R_2nd ENABLE
// ======================== ENABLE ==========================
; L159
LOAD      M04100	// R_P&P_10 Y Pos.1st IDLE
AND       P0005D	// R_P&P UP (SENSOR)
OUT       M13190	// R_2nd MAND PICKER ENABLE
; L160
LOAD      M04102	// R_P&P_10 Y Pos.3rd PLACE
AND       P0005E	// R_P&P DOWN
AND       P00163	// R_P&P 2nd EJECT OFF
OR        M13192	// R_2nd MAND AUAc ¥ìe¨úi¢¯E
AND NOT   M03101	// R_P&P_10 Y PICKUP POS ->
AND NOT   M03102	// R_P&P_10 Y PUT POS ->
AND NOT   M1309A	// R_2nd MAND ORIGIN KP
AND NOT   M0000A	// DRY RUN OFF PLS
OUT       M13192	// R_2nd MAND AUAc ¥ìe¨úi¢¯E
; L162
LOAD      M04101	// R_P&P_10 Y Pos.2nd PICK
AND       P0005E	// R_P&P DOWN
AND       P00164	// R_P&P 3rd EJECT ON
OR        M13194	// R_2nd MAND AUAc ¡Æ¢®A¢ç¡Æ¡§
AND NOT   M03100	// R_P&P_10 Y IDLE POS ->
AND NOT   M03101	// R_P&P_10 Y PICKUP POS ->
AND NOT   M03102	// R_P&P_10 Y PUT POS ->
AND NOT   M1309A	// R_2nd MAND ORIGIN KP
AND NOT   M0000A	// DRY RUN OFF PLS
OUT       M13194	// R_2nd MAND AUAc ¡Æ¢®A¢ç¡Æ¡§
; L164
LOAD NOT  M01421	// R_PP 2 VC KP
AND NOT   M06612	// R_2nd DET VAC ON
AND       M13080	// R_2nd MAND CYCLE RUN
ANDP      P0005D	// R_P&P UP (SENSOR)
AND       M04102	// R_P&P_10 Y Pos.3rd PLACE
AND NOT   M1902F	// DRY RUN
OUT       M1319F	// R_2nd MAND AUAc ¨ú©ª¨úiAu
// ======================== TIMER ==========================
; L166
LOAD      P00087	// R_2nd SS CLAMP.L UP
AND NOT   P00088	// R_2nd SS CLAMP.L DN
TON       T4220 15	// R_2nd SS CLAMP.L UP
; L167
LOAD      P00088	// R_2nd SS CLAMP.L DN
AND NOT   P00087	// R_2nd SS CLAMP.L UP
TON       T4221 15	// R_2nd SS CLAMP.L DN
; L168
LOAD      P00085	// R_2nd SS CLAMP.R UP
AND NOT   P00086	// R_2nd SS CLAMP.R DN
TON       T4222 15	// R_2nd SS CLAMP.R UP

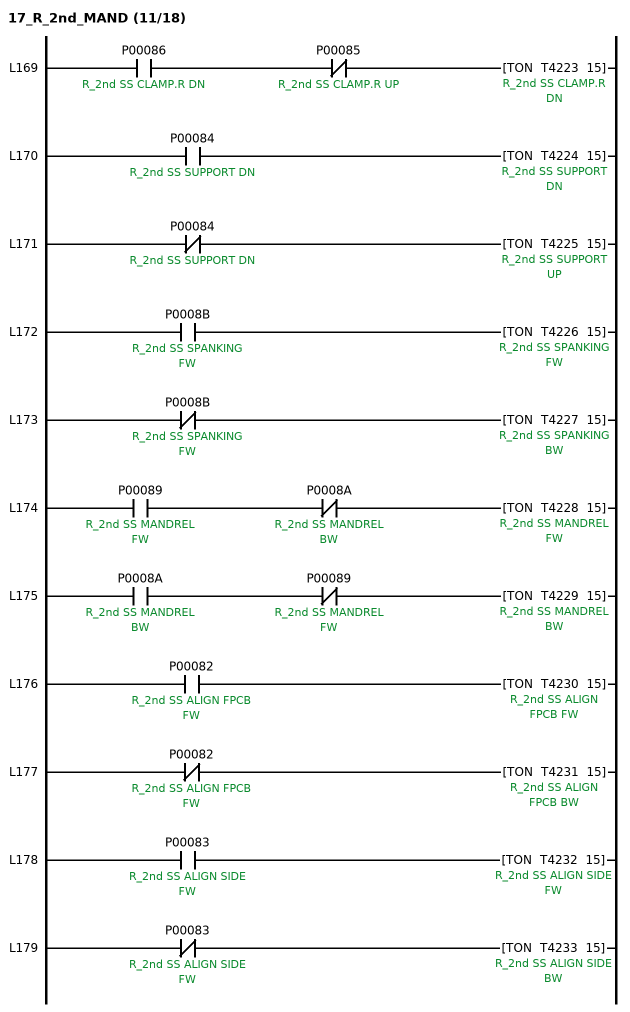
; L169
LOAD      P00086	// R_2nd SS CLAMP.R DN
AND NOT   P00085	// R_2nd SS CLAMP.R UP
TON       T4223 15	// R_2nd SS CLAMP.R DN
; L170
LOAD      P00084	// R_2nd SS SUPPORT DN
TON       T4224 15	// R_2nd SS SUPPORT DN
; L171
LOAD NOT  P00084	// R_2nd SS SUPPORT DN
TON       T4225 15	// R_2nd SS SUPPORT UP
; L172
LOAD      P0008B	// R_2nd SS SPANKING FW
TON       T4226 15	// R_2nd SS SPANKING FW
; L173
LOAD NOT  P0008B	// R_2nd SS SPANKING FW
TON       T4227 15	// R_2nd SS SPANKING BW
; L174
LOAD      P00089	// R_2nd SS MANDREL FW
AND NOT   P0008A	// R_2nd SS MANDREL BW
TON       T4228 15	// R_2nd SS MANDREL FW
; L175
LOAD      P0008A	// R_2nd SS MANDREL BW
AND NOT   P00089	// R_2nd SS MANDREL FW
TON       T4229 15	// R_2nd SS MANDREL BW
; L176
LOAD      P00082	// R_2nd SS ALIGN FPCB FW
TON       T4230 15	// R_2nd SS ALIGN FPCB FW
; L177
LOAD NOT  P00082	// R_2nd SS ALIGN FPCB FW
TON       T4231 15	// R_2nd SS ALIGN FPCB BW
; L178
LOAD      P00083	// R_2nd SS ALIGN SIDE FW
TON       T4232 15	// R_2nd SS ALIGN SIDE FW
; L179
LOAD NOT  P00083	// R_2nd SS ALIGN SIDE FW
TON       T4233 15	// R_2nd SS ALIGN SIDE BW

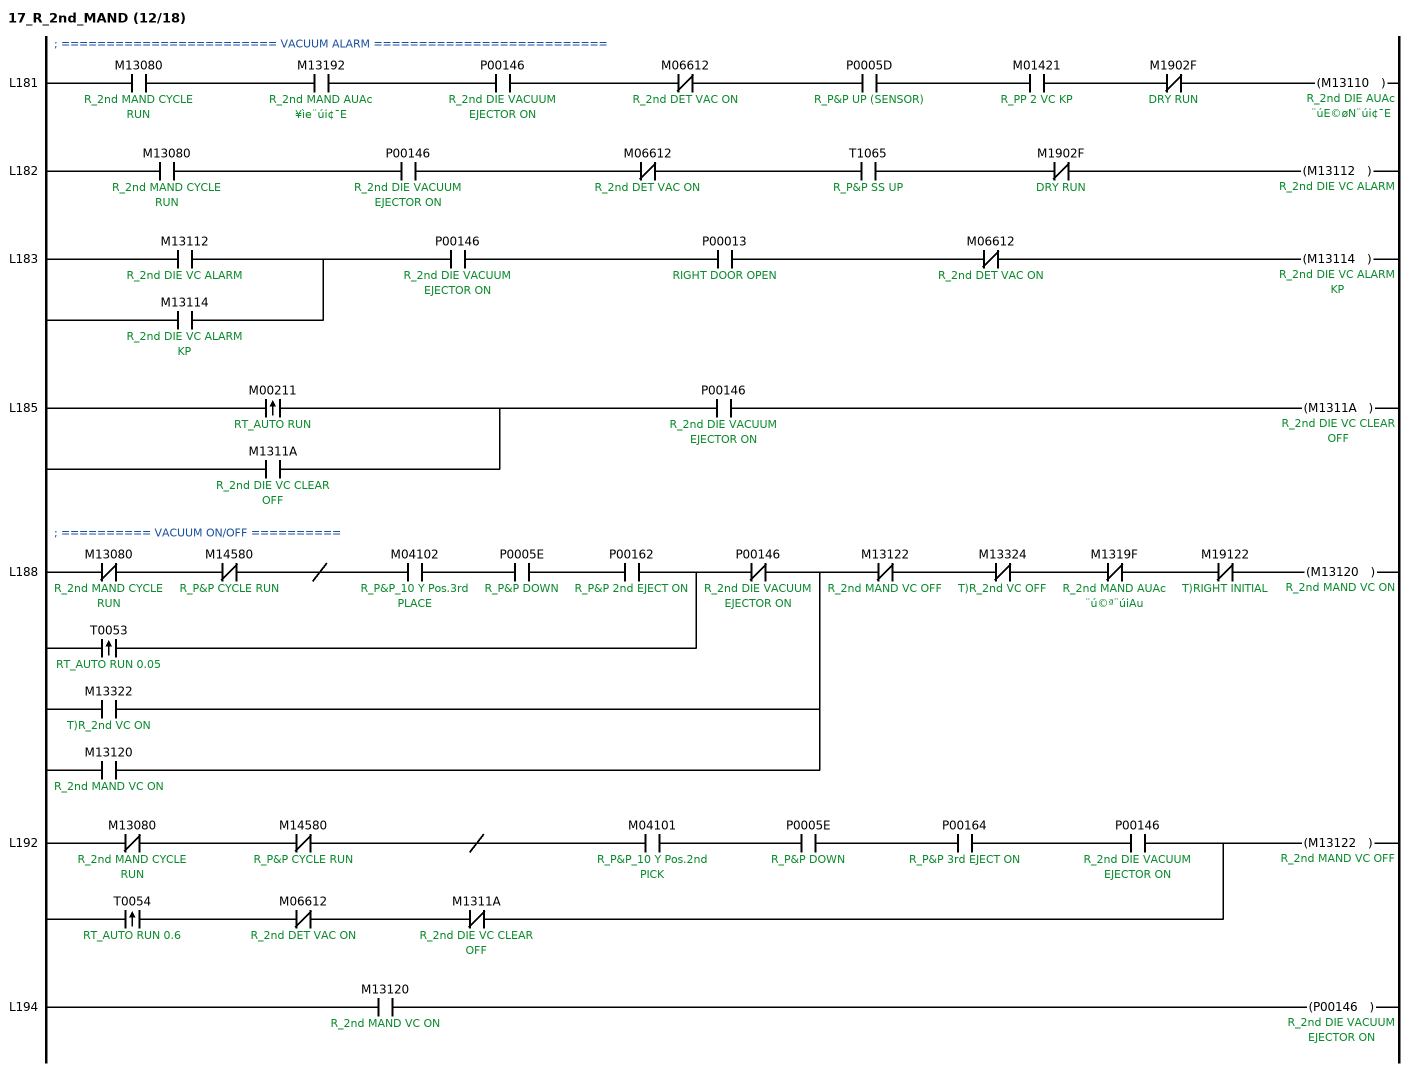
// ======================== VACUUM ALARM ==========================
; L181
LOAD      M13080	// R_2nd MAND CYCLE RUN
AND       M13192	// R_2nd MAND AUAc ¥ìe¨úi¢¯E
AND       P00146	// R_2nd DIE VACUUM EJECTOR ON
AND NOT   M06612	// R_2nd DET VAC ON
AND       P0005D	// R_P&P UP (SENSOR)
AND       M01421	// R_PP 2 VC KP
AND NOT   M1902F	// DRY RUN
OUT       M13110	// R_2nd DIE AUAc ¨úE©øN¨úi¢¯E
; L182
LOAD      M13080	// R_2nd MAND CYCLE RUN
AND       P00146	// R_2nd DIE VACUUM EJECTOR ON
AND NOT   M06612	// R_2nd DET VAC ON
AND       T1065	// R_P&P SS UP
AND NOT   M1902F	// DRY RUN
OUT       M13112	// R_2nd DIE VC ALARM
; L183
LOAD      M13112	// R_2nd DIE VC ALARM
OR        M13114	// R_2nd DIE VC ALARM KP
AND       P00146	// R_2nd DIE VACUUM EJECTOR ON
AND       P00013	// RIGHT DOOR OPEN
AND NOT   M06612	// R_2nd DET VAC ON
OUT       M13114	// R_2nd DIE VC ALARM KP
; L185
LOADP     M00211	// RT_AUTO RUN
OR        M1311A	// R_2nd DIE VC CLEAR OFF
AND       P00146	// R_2nd DIE VACUUM EJECTOR ON
OUT       M1311A	// R_2nd DIE VC CLEAR OFF
// ========== VACUUM ON/OFF ==========
; L188
LOAD NOT  M13080	// R_2nd MAND CYCLE RUN
AND NOT   M14580	// R_P&P CYCLE RUN
NOT
AND       M04102	// R_P&P_10 Y Pos.3rd PLACE
AND       P0005E	// R_P&P DOWN
AND       P00162	// R_P&P 2nd EJECT ON
ORP       T0053	// RT_AUTO RUN 0.05
AND NOT   P00146	// R_2nd DIE VACUUM EJECTOR ON
OR        M13322	// T)R_2nd VC ON
OR        M13120	// R_2nd MAND VC ON
AND NOT   M13122	// R_2nd MAND VC OFF
AND NOT   M13324	// T)R_2nd VC OFF
AND NOT   M1319F	// R_2nd MAND AUAc ¨ú©ª¨úiAu
AND NOT   M19122	// T)RIGHT INITIAL
OUT       M13120	// R_2nd MAND VC ON
; L192
LOAD NOT  M13080	// R_2nd MAND CYCLE RUN
AND NOT   M14580	// R_P&P CYCLE RUN
NOT
AND       M04101	// R_P&P_10 Y Pos.2nd PICK
AND       P0005E	// R_P&P DOWN
AND       P00164	// R_P&P 3rd EJECT ON
AND       P00146	// R_2nd DIE VACUUM EJECTOR ON
LOADP     T0054	// RT_AUTO RUN 0.6
AND NOT   M06612	// R_2nd DET VAC ON
AND NOT   M1311A	// R_2nd DIE VC CLEAR OFF
OR LOAD
OUT       M13122	// R_2nd MAND VC OFF
; L194
LOAD      M13120	// R_2nd MAND VC ON
OUT       P00146	// R_2nd DIE VACUUM EJECTOR ON

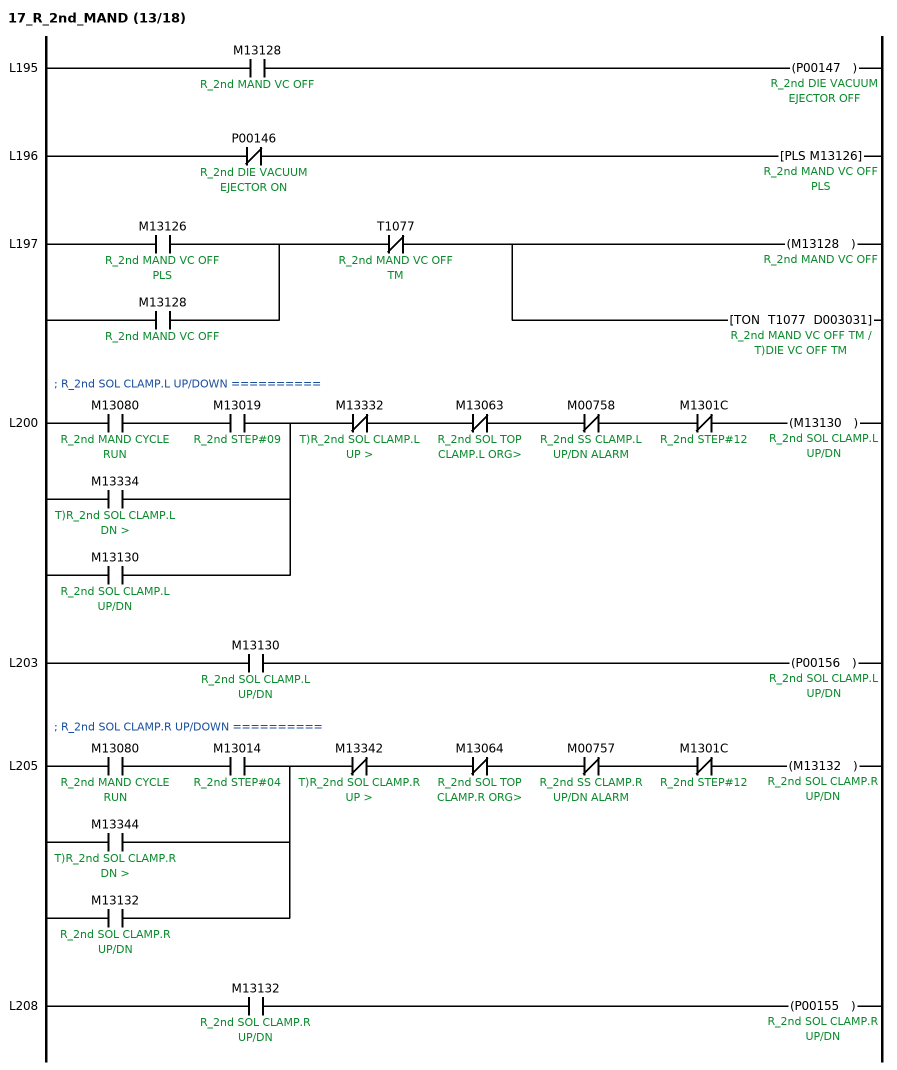
; L195
LOAD      M13128	// R_2nd MAND VC OFF
OUT       P00147	// R_2nd DIE VACUUM EJECTOR OFF
; L196
LOAD NOT  P00146	// R_2nd DIE VACUUM EJECTOR ON
OUTP      M13126	// R_2nd MAND VC OFF PLS
; L197
LOAD      M13126	// R_2nd MAND VC OFF PLS
OR        M13128	// R_2nd MAND VC OFF
AND NOT   T1077	// R_2nd MAND VC OFF TM
OUT       M13128	// R_2nd MAND VC OFF
TON       T1077 D003031	// R_2nd MAND VC OFF TM / T)DIE VC OFF TM
//  R_2nd SOL CLAMP.L UP/DOWN ==========
; L200
LOAD      M13080	// R_2nd MAND CYCLE RUN
AND       M13019	// R_2nd STEP#09
OR        M13334	// T)R_2nd SOL CLAMP.L DN >
OR        M13130	// R_2nd SOL CLAMP.L UP/DN
AND NOT   M13332	// T)R_2nd SOL CLAMP.L UP >
AND NOT   M13063	// R_2nd SOL TOP CLAMP.L ORG>
AND NOT   M00758	// R_2nd SS CLAMP.L UP/DN ALARM
AND NOT   M1301C	// R_2nd STEP#12
OUT       M13130	// R_2nd SOL CLAMP.L UP/DN
; L203
LOAD      M13130	// R_2nd SOL CLAMP.L UP/DN
OUT       P00156	// R_2nd SOL CLAMP.L UP/DN
//  R_2nd SOL CLAMP.R UP/DOWN ==========
; L205
LOAD      M13080	// R_2nd MAND CYCLE RUN
AND       M13014	// R_2nd STEP#04
OR        M13344	// T)R_2nd SOL CLAMP.R DN >
OR        M13132	// R_2nd SOL CLAMP.R UP/DN
AND NOT   M13342	// T)R_2nd SOL CLAMP.R UP >
AND NOT   M13064	// R_2nd SOL TOP CLAMP.R ORG>
AND NOT   M00757	// R_2nd SS CLAMP.R UP/DN ALARM
AND NOT   M1301C	// R_2nd STEP#12
OUT       M13132	// R_2nd SOL CLAMP.R UP/DN
; L208
LOAD      M13132	// R_2nd SOL CLAMP.R UP/DN
OUT       P00155	// R_2nd SOL CLAMP.R UP/DN

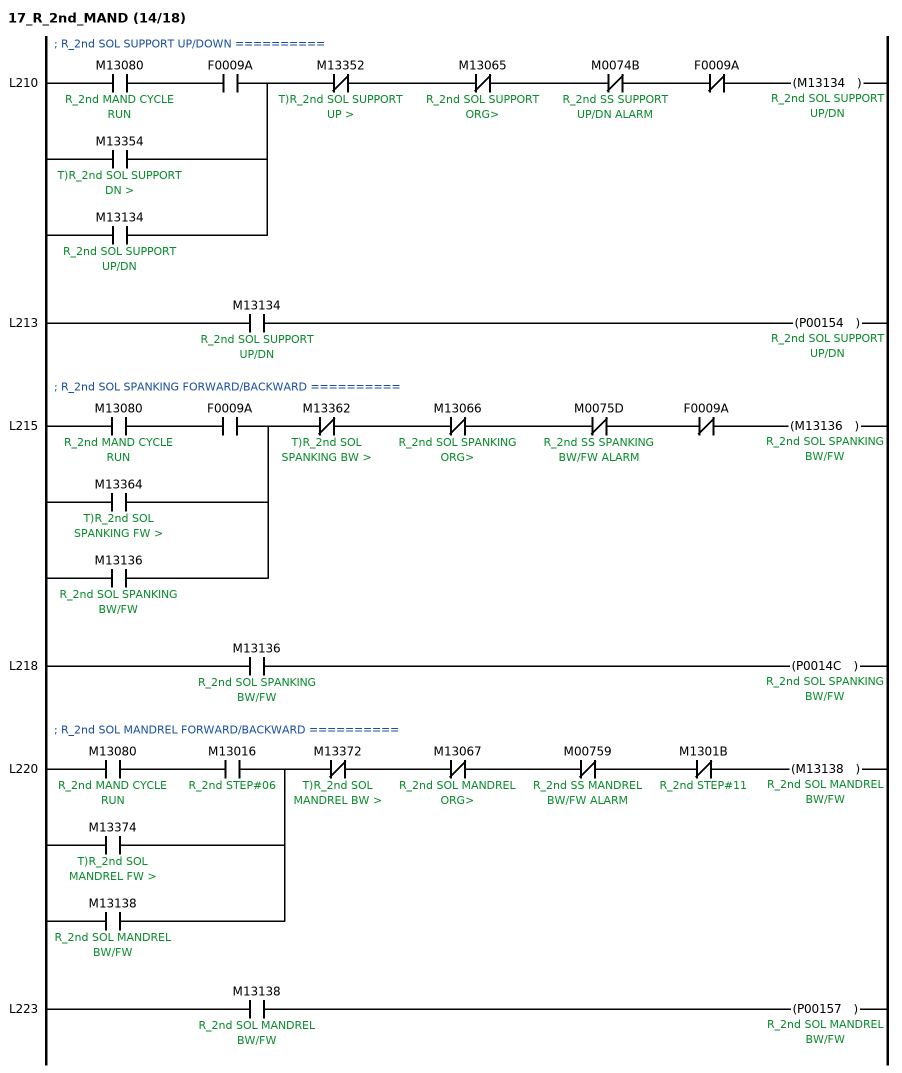
// R_2nd SOL SUPPORT UP/DOWN ==========
; L210
LOAD      M13080	// R_2nd MAND CYCLE RUN
AND       F0009A
OR        M13354	// T)R_2nd SOL SUPPORT DN >
OR        M13134	// R_2nd SOL SUPPORT UP/DN
AND NOT   M13352	// T)R_2nd SOL SUPPORT UP >
AND NOT   M13065	// R_2nd SOL SUPPORT ORG>
AND NOT   M0074B	// R_2nd SS SUPPORT UP/DN ALARM
AND NOT   F0009A
OUT       M13134	// R_2nd SOL SUPPORT UP/DN
; L213
LOAD      M13134	// R_2nd SOL SUPPORT UP/DN
OUT       P00154	// R_2nd SOL SUPPORT UP/DN
// R_2nd SOL SPANKING FORWARD/BACKWARD ==========
; L215
LOAD      M13080	// R_2nd MAND CYCLE RUN
AND       F0009A
OR        M13364	// T)R_2nd SOL SPANKING FW >
OR        M13136	// R_2nd SOL SPANKING BW/FW
AND NOT   M13362	// T)R_2nd SOL SPANKING BW >
AND NOT   M13066	// R_2nd SOL SPANKING ORG>
AND NOT   M0075D	// R_2nd SS SPANKING BW/FW ALARM
AND NOT   F0009A
OUT       M13136	// R_2nd SOL SPANKING BW/FW
; L218
LOAD      M13136	// R_2nd SOL SPANKING BW/FW
OUT       P0014C	// R_2nd SOL SPANKING BW/FW
// R_2nd SOL MANDREL FORWARD/BACKWARD ==========
; L220
LOAD      M13080	// R_2nd MAND CYCLE RUN
AND       M13016	// R_2nd STEP#06
OR        M13374	// T)R_2nd SOL MANDREL FW >
OR        M13138	// R_2nd SOL MANDREL BW/FW
AND NOT   M13372	// T)R_2nd SOL MANDREL BW >
AND NOT   M13067	// R_2nd SOL MANDREL ORG>
AND NOT   M00759	// R_2nd SS MANDREL BW/FW ALARM
AND NOT   M1301B	// R_2nd STEP#11
OUT       M13138	// R_2nd SOL MANDREL BW/FW
; L223
LOAD      M13138	// R_2nd SOL MANDREL BW/FW
OUT       P00157	// R_2nd SOL MANDREL BW/FW

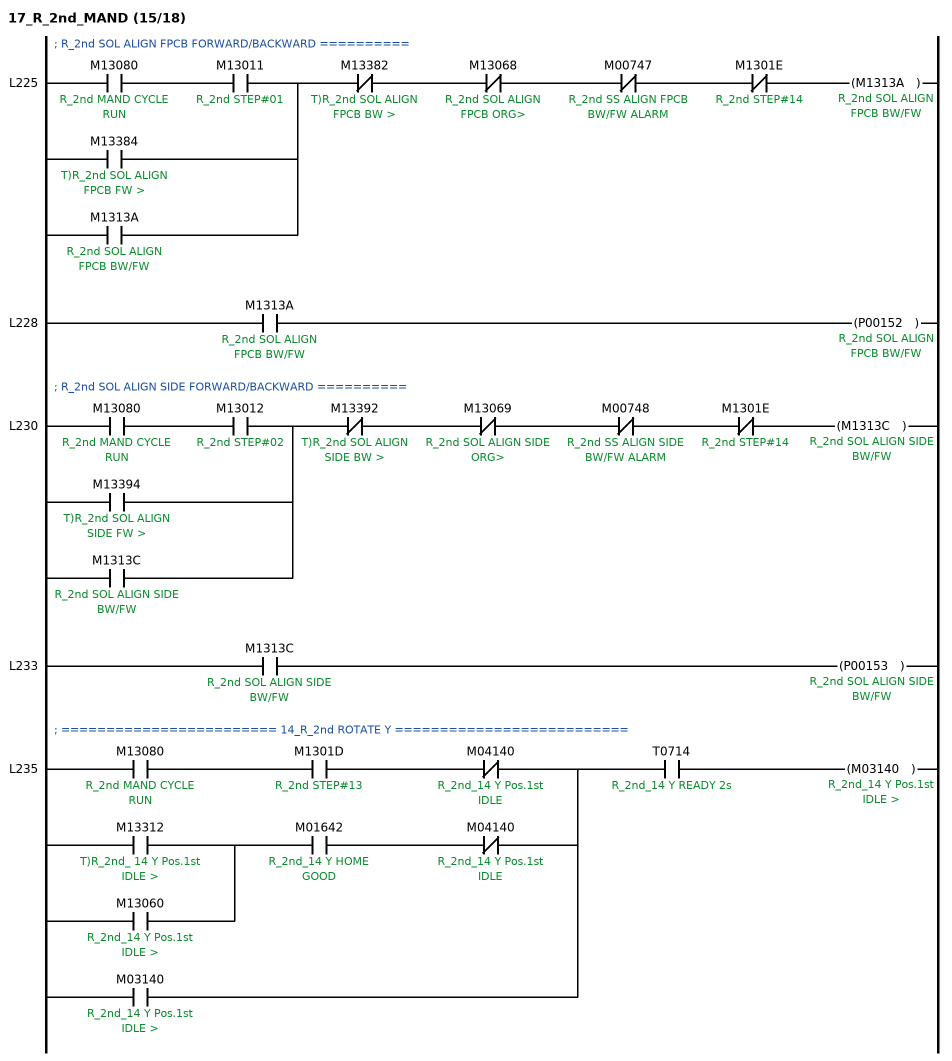
// R_2nd SOL ALIGN FPCB FORWARD/BACKWARD ==========
; L225
LOAD      M13080	// R_2nd MAND CYCLE RUN
AND       M13011	// R_2nd STEP#01
OR        M13384	// T)R_2nd SOL ALIGN FPCB FW >
OR        M1313A	// R_2nd SOL ALIGN FPCB BW/FW
AND NOT   M13382	// T)R_2nd SOL ALIGN FPCB BW >
AND NOT   M13068	// R_2nd SOL ALIGN FPCB ORG>
AND NOT   M00747	// R_2nd SS ALIGN FPCB BW/FW ALARM
AND NOT   M1301E	// R_2nd STEP#14
OUT       M1313A	// R_2nd SOL ALIGN FPCB BW/FW
; L228
LOAD      M1313A	// R_2nd SOL ALIGN FPCB BW/FW
OUT       P00152	// R_2nd SOL ALIGN FPCB BW/FW
// R_2nd SOL ALIGN SIDE FORWARD/BACKWARD ==========
; L230
LOAD      M13080	// R_2nd MAND CYCLE RUN
AND       M13012	// R_2nd STEP#02
OR        M13394	// T)R_2nd SOL ALIGN SIDE FW >
OR        M1313C	// R_2nd SOL ALIGN SIDE BW/FW
AND NOT   M13392	// T)R_2nd SOL ALIGN SIDE BW >
AND NOT   M13069	// R_2nd SOL ALIGN SIDE ORG>
AND NOT   M00748	// R_2nd SS ALIGN SIDE BW/FW ALARM
AND NOT   M1301E	// R_2nd STEP#14
OUT       M1313C	// R_2nd SOL ALIGN SIDE BW/FW
; L233
LOAD      M1313C	// R_2nd SOL ALIGN SIDE BW/FW
OUT       P00153	// R_2nd SOL ALIGN SIDE BW/FW
// ======================== 14_R_2nd ROTATE Y ==========================
; L235
LOAD      M13080	// R_2nd MAND CYCLE RUN
AND       M1301D	// R_2nd STEP#13
AND NOT   M04140	// R_2nd_14 Y Pos.1st IDLE
LOAD      M13312	// T)R_2nd_ 14 Y Pos.1st IDLE >
OR        M13060	// R_2nd_14 Y Pos.1st IDLE >
AND       M01642	// R_2nd_14 Y HOME GOOD
AND NOT   M04140	// R_2nd_14 Y Pos.1st IDLE
OR LOAD
OR        M03140	// R_2nd_14 Y Pos.1st IDLE >
AND       T0714	// R_2nd_14 Y READY 2s
OUT       M03140	// R_2nd_14 Y Pos.1st IDLE >

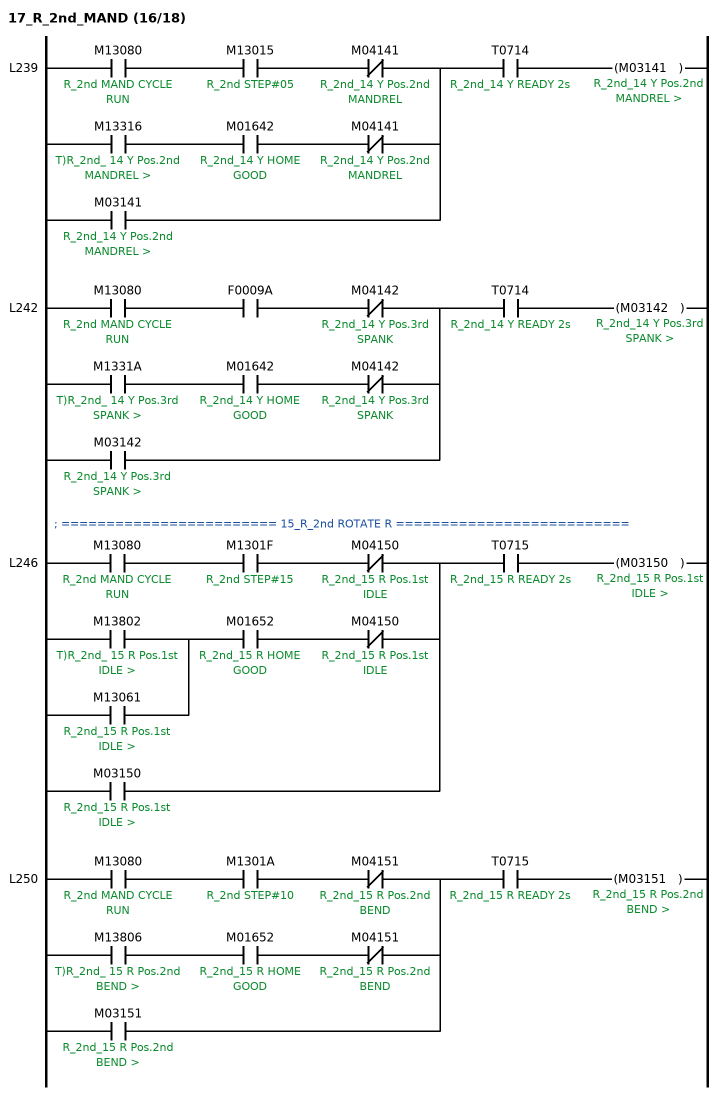
; L239
LOAD      M13080	// R_2nd MAND CYCLE RUN
AND       M13015	// R_2nd STEP#05
AND NOT   M04141	// R_2nd_14 Y Pos.2nd MANDREL
LOAD      M13316	// T)R_2nd_ 14 Y Pos.2nd MANDREL >
AND       M01642	// R_2nd_14 Y HOME GOOD
AND NOT   M04141	// R_2nd_14 Y Pos.2nd MANDREL
OR LOAD
OR        M03141	// R_2nd_14 Y Pos.2nd MANDREL >
AND       T0714	// R_2nd_14 Y READY 2s
OUT       M03141	// R_2nd_14 Y Pos.2nd MANDREL >
; L242
LOAD      M13080	// R_2nd MAND CYCLE RUN
AND       F0009A
AND NOT   M04142	// R_2nd_14 Y Pos.3rd SPANK
LOAD      M1331A	// T)R_2nd_ 14 Y Pos.3rd SPANK >
AND       M01642	// R_2nd_14 Y HOME GOOD
AND NOT   M04142	// R_2nd_14 Y Pos.3rd SPANK
OR LOAD
OR        M03142	// R_2nd_14 Y Pos.3rd SPANK >
AND       T0714	// R_2nd_14 Y READY 2s
OUT       M03142	// R_2nd_14 Y Pos.3rd SPANK >
// ======================== 15_R_2nd ROTATE R ==========================
; L246
LOAD      M13080	// R_2nd MAND CYCLE RUN
AND       M1301F	// R_2nd STEP#15
AND NOT   M04150	// R_2nd_15 R Pos.1st IDLE
LOAD      M13802	// T)R_2nd_ 15 R Pos.1st IDLE >
OR        M13061	// R_2nd_15 R Pos.1st IDLE >
AND       M01652	// R_2nd_15 R HOME GOOD
AND NOT   M04150	// R_2nd_15 R Pos.1st IDLE
OR LOAD
OR        M03150	// R_2nd_15 R Pos.1st IDLE >
AND       T0715	// R_2nd_15 R READY 2s
OUT       M03150	// R_2nd_15 R Pos.1st IDLE >
; L250
LOAD      M13080	// R_2nd MAND CYCLE RUN
AND       M1301A	// R_2nd STEP#10
AND NOT   M04151	// R_2nd_15 R Pos.2nd BEND
LOAD      M13806	// T)R_2nd_ 15 R Pos.2nd BEND >
AND       M01652	// R_2nd_15 R HOME GOOD
AND NOT   M04151	// R_2nd_15 R Pos.2nd BEND
OR LOAD
OR        M03151	// R_2nd_15 R Pos.2nd BEND >
AND       T0715	// R_2nd_15 R READY 2s
OUT       M03151	// R_2nd_15 R Pos.2nd BEND >

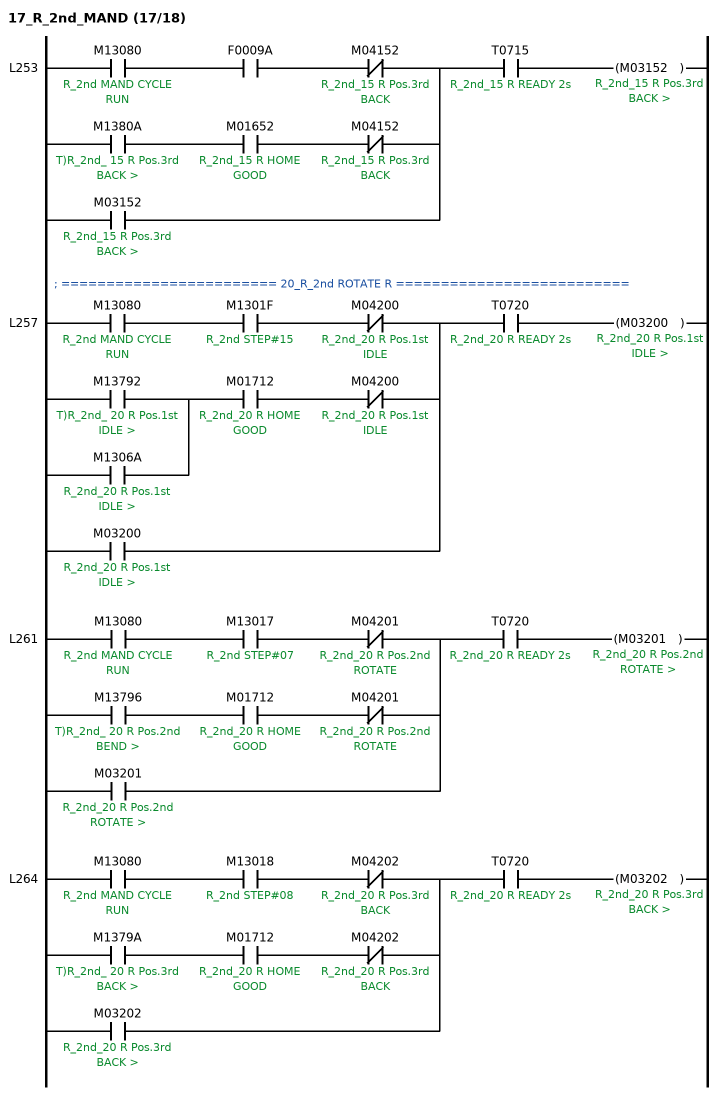
; L253
LOAD      M13080	// R_2nd MAND CYCLE RUN
AND       F0009A
AND NOT   M04152	// R_2nd_15 R Pos.3rd BACK
LOAD      M1380A	// T)R_2nd_ 15 R Pos.3rd BACK >
AND       M01652	// R_2nd_15 R HOME GOOD
AND NOT   M04152	// R_2nd_15 R Pos.3rd BACK
OR LOAD
OR        M03152	// R_2nd_15 R Pos.3rd BACK >
AND       T0715	// R_2nd_15 R READY 2s
OUT       M03152	// R_2nd_15 R Pos.3rd BACK >
// ======================== 20_R_2nd ROTATE R ==========================
; L257
LOAD      M13080	// R_2nd MAND CYCLE RUN
AND       M1301F	// R_2nd STEP#15
AND NOT   M04200	// R_2nd_20 R Pos.1st IDLE
LOAD      M13792	// T)R_2nd_ 20 R Pos.1st IDLE >
OR        M1306A	// R_2nd_20 R Pos.1st IDLE >
AND       M01712	// R_2nd_20 R HOME GOOD
AND NOT   M04200	// R_2nd_20 R Pos.1st IDLE
OR LOAD
OR        M03200	// R_2nd_20 R Pos.1st IDLE >
AND       T0720	// R_2nd_20 R READY 2s
OUT       M03200	// R_2nd_20 R Pos.1st IDLE >
; L261
LOAD      M13080	// R_2nd MAND CYCLE RUN
AND       M13017	// R_2nd STEP#07
AND NOT   M04201	// R_2nd_20 R Pos.2nd ROTATE
LOAD      M13796	// T)R_2nd_ 20 R Pos.2nd BEND >
AND       M01712	// R_2nd_20 R HOME GOOD
AND NOT   M04201	// R_2nd_20 R Pos.2nd ROTATE
OR LOAD
OR        M03201	// R_2nd_20 R Pos.2nd ROTATE >
AND       T0720	// R_2nd_20 R READY 2s
OUT       M03201	// R_2nd_20 R Pos.2nd ROTATE >
; L264
LOAD      M13080	// R_2nd MAND CYCLE RUN
AND       M13018	// R_2nd STEP#08
AND NOT   M04202	// R_2nd_20 R Pos.3rd BACK
LOAD      M1379A	// T)R_2nd_ 20 R Pos.3rd BACK >
AND       M01712	// R_2nd_20 R HOME GOOD
AND NOT   M04202	// R_2nd_20 R Pos.3rd BACK
OR LOAD
OR        M03202	// R_2nd_20 R Pos.3rd BACK >
AND       T0720	// R_2nd_20 R READY 2s
OUT       M03202	// R_2nd_20 R Pos.3rd BACK >

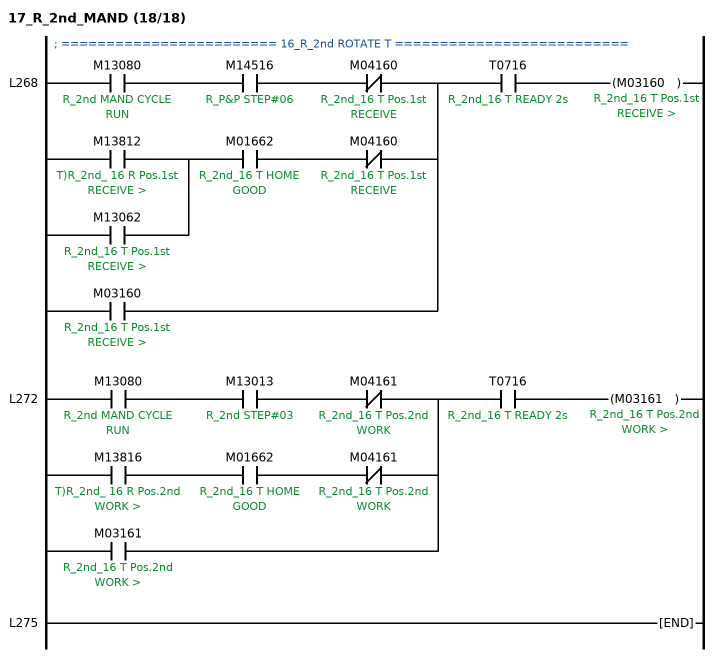
// ======================== 16_R_2nd ROTATE T ==========================
; L268
LOAD      M13080	// R_2nd MAND CYCLE RUN
AND       M14516	// R_P&P STEP#06
AND NOT   M04160	// R_2nd_16 T Pos.1st RECEIVE
LOAD      M13812	// T)R_2nd_ 16 R Pos.1st RECEIVE >
OR        M13062	// R_2nd_16 T Pos.1st RECEIVE >
AND       M01662	// R_2nd_16 T HOME GOOD
AND NOT   M04160	// R_2nd_16 T Pos.1st RECEIVE
OR LOAD
OR        M03160	// R_2nd_16 T Pos.1st RECEIVE >
AND       T0716	// R_2nd_16 T READY 2s
OUT       M03160	// R_2nd_16 T Pos.1st RECEIVE >
; L272
LOAD      M13080	// R_2nd MAND CYCLE RUN
AND       M13013	// R_2nd STEP#03
AND NOT   M04161	// R_2nd_16 T Pos.2nd WORK
LOAD      M13816	// T)R_2nd_ 16 R Pos.2nd WORK >
AND       M01662	// R_2nd_16 T HOME GOOD
AND NOT   M04161	// R_2nd_16 T Pos.2nd WORK
OR LOAD
OR        M03161	// R_2nd_16 T Pos.2nd WORK >
AND       T0716	// R_2nd_16 T READY 2s
OUT       M03161	// R_2nd_16 T Pos.2nd WORK >
; L275
END

PROGRAM 18_R_3rd_MAND (task: ¨ö¨¬A¥ì CA¡¤I¡¾¡¿¡¤¡Í)

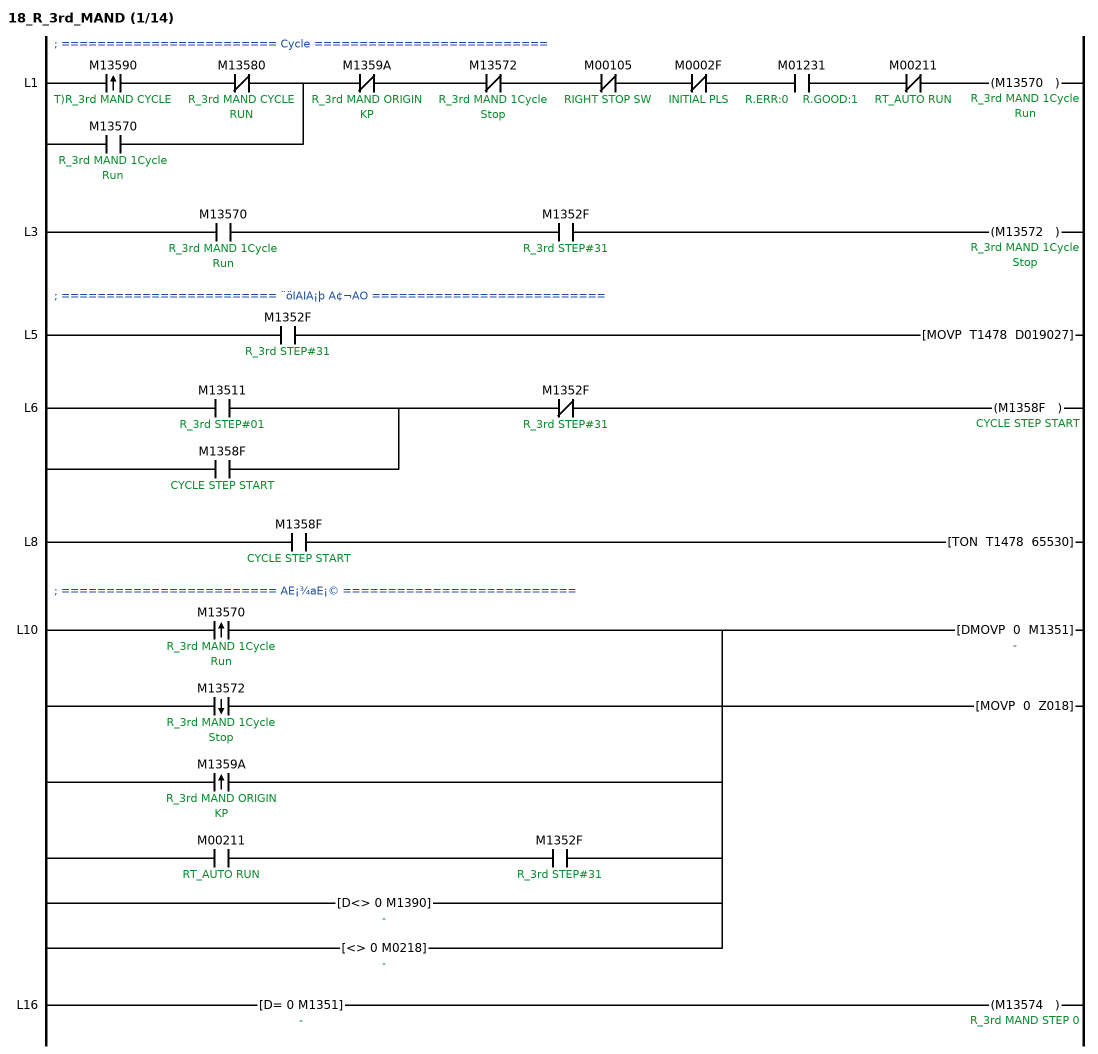
// ======================== Cycle ==========================
; L1
LOADP     M13590	// T)R_3rd MAND CYCLE
AND NOT   M13580	// R_3rd MAND CYCLE RUN
OR        M13570	// R_3rd MAND 1Cycle Run
AND NOT   M1359A	// R_3rd MAND ORIGIN KP
AND NOT   M13572	// R_3rd MAND 1Cycle Stop
AND NOT   M00105	// RIGHT STOP SW
AND NOT   M0002F	// INITIAL PLS
AND       M01231	// R.ERR:0    R.GOOD:1
AND NOT   M00211	// RT_AUTO RUN
OUT       M13570	// R_3rd MAND 1Cycle Run
; L3
LOAD      M13570	// R_3rd MAND 1Cycle Run
AND       M1352F	// R_3rd STEP#31
OUT       M13572	// R_3rd MAND 1Cycle Stop
// ======================== ¨öIAIA¡þ A¢¬AO ==========================
; L5
LOAD      M1352F	// R_3rd STEP#31
MOVP      T1478 D019027
; L6
LOAD      M13511	// R_3rd STEP#01
OR        M1358F	// CYCLE STEP START
AND NOT   M1352F	// R_3rd STEP#31
OUT       M1358F	// CYCLE STEP START
; L8
LOAD      M1358F	// CYCLE STEP START
TON       T1478 65530
// ======================== AE¡¾aE¡© ==========================
; L10
LOADP     M13570	// R_3rd MAND 1Cycle Run
ORN       M13572	// R_3rd MAND 1Cycle Stop
ORP       M1359A	// R_3rd MAND ORIGIN KP
LOAD      M00211	// RT_AUTO RUN
AND       M1352F	// R_3rd STEP#31
OR LOAD
ORD<>     0 M1390	// -
OR<>      0 M0218	// -
DMOVP     0 M1351	// -
MOVP      0 Z018
; L16
LOADD=    0 M1351	// -
OUT       M13574	// R_3rd MAND STEP 0

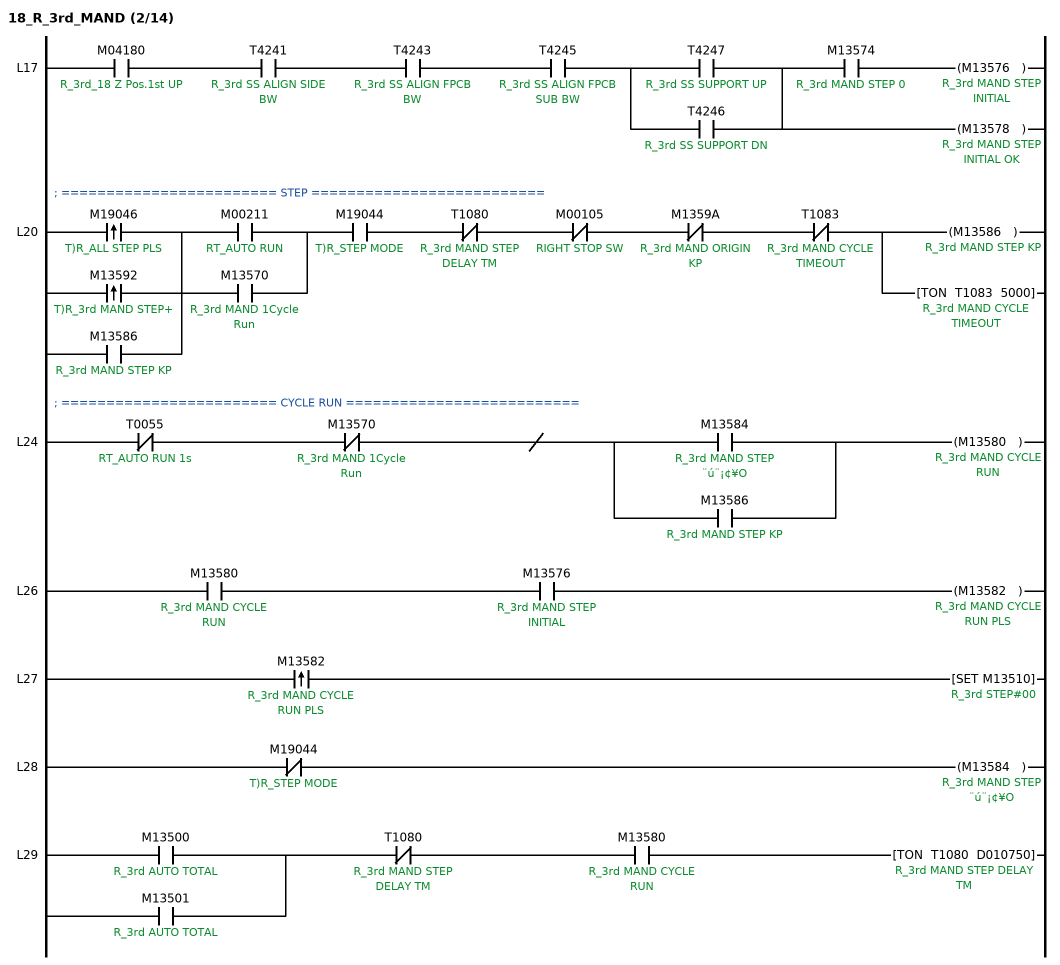
; L17
LOAD      M04180	// R_3rd_18 Z Pos.1st UP
AND       T4241	// R_3rd SS ALIGN SIDE BW
AND       T4243	// R_3rd SS ALIGN FPCB BW
AND       T4245	// R_3rd SS ALIGN FPCB SUB BW
LOAD      T4247	// R_3rd SS SUPPORT UP
OR        T4246	// R_3rd SS SUPPORT DN
AND LOAD
MPUSH
AND       M13574	// R_3rd MAND STEP 0
OUT       M13576	// R_3rd MAND STEP INITIAL
MPOP
OUT       M13578	// R_3rd MAND STEP INITIAL OK
// ======================== STEP ==========================
; L20
LOADP     M19046	// T)R_ALL STEP PLS
ORP       M13592	// T)R_3rd MAND STEP+
OR        M13586	// R_3rd MAND STEP KP
LOAD      M00211	// RT_AUTO RUN
OR        M13570	// R_3rd MAND 1Cycle Run
AND LOAD
AND       M19044	// T)R_STEP MODE
AND NOT   T1080	// R_3rd MAND STEP DELAY TM
AND NOT   M00105	// RIGHT STOP SW
AND NOT   M1359A	// R_3rd MAND ORIGIN KP
AND NOT   T1083	// R_3rd MAND CYCLE TIMEOUT
OUT       M13586	// R_3rd MAND STEP KP
TON       T1083 5000	// R_3rd MAND CYCLE TIMEOUT
// ======================== CYCLE RUN ==========================
; L24
LOAD NOT  T0055	// RT_AUTO RUN 1s
AND NOT   M13570	// R_3rd MAND 1Cycle Run
NOT
LOAD      M13584	// R_3rd MAND STEP ¨ú¨¡¢¥O
OR        M13586	// R_3rd MAND STEP KP
AND LOAD
OUT       M13580	// R_3rd MAND CYCLE RUN
; L26
LOAD      M13580	// R_3rd MAND CYCLE RUN
AND       M13576	// R_3rd MAND STEP INITIAL
OUT       M13582	// R_3rd MAND CYCLE RUN PLS
; L27
LOADP     M13582	// R_3rd MAND CYCLE RUN PLS
SET       M13510	// R_3rd STEP#00
; L28
LOAD NOT  M19044	// T)R_STEP MODE
OUT       M13584	// R_3rd MAND STEP ¨ú¨¡¢¥O
; L29
LOAD      M13500	// R_3rd AUTO TOTAL
OR        M13501	// R_3rd AUTO TOTAL
AND NOT   T1080	// R_3rd MAND STEP DELAY TM
AND       M13580	// R_3rd MAND CYCLE RUN
TON       T1080 D010750	// R_3rd MAND STEP DELAY TM

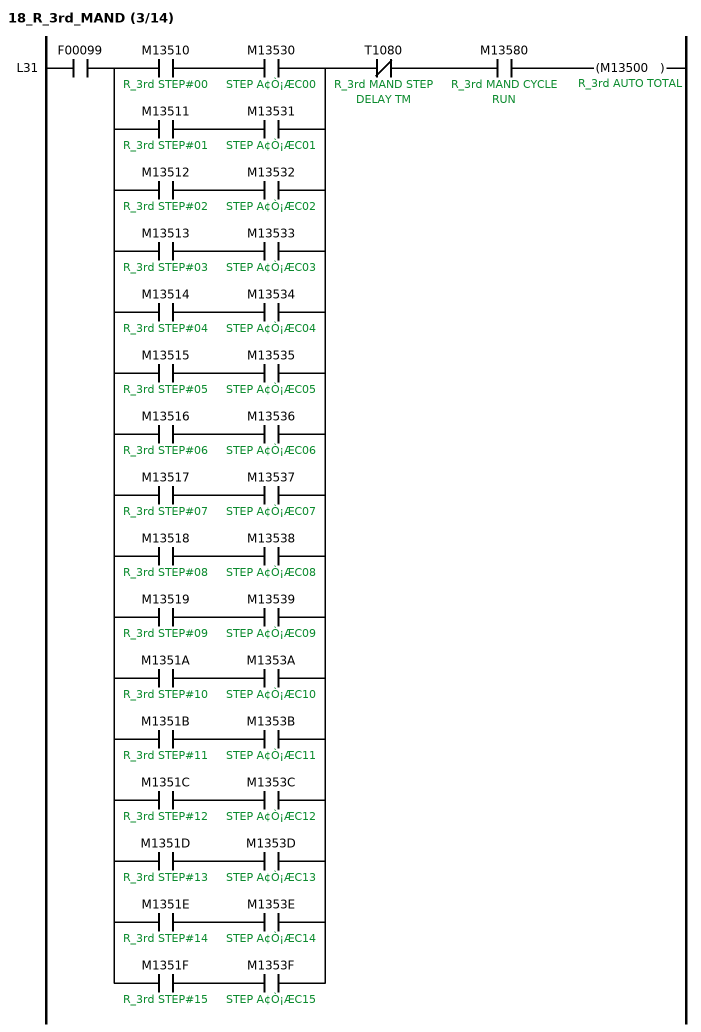
; L31
LOAD      F00099
LOAD      M13510	// R_3rd STEP#00
AND       M13530	// STEP A¢Ò¡ÆC00
LOAD      M13511	// R_3rd STEP#01
AND       M13531	// STEP A¢Ò¡ÆC01
OR LOAD
LOAD      M13512	// R_3rd STEP#02
AND       M13532	// STEP A¢Ò¡ÆC02
OR LOAD
LOAD      M13513	// R_3rd STEP#03
AND       M13533	// STEP A¢Ò¡ÆC03
OR LOAD
LOAD      M13514	// R_3rd STEP#04
AND       M13534	// STEP A¢Ò¡ÆC04
OR LOAD
LOAD      M13515	// R_3rd STEP#05
AND       M13535	// STEP A¢Ò¡ÆC05
OR LOAD
LOAD      M13516	// R_3rd STEP#06
AND       M13536	// STEP A¢Ò¡ÆC06
OR LOAD
LOAD      M13517	// R_3rd STEP#07
AND       M13537	// STEP A¢Ò¡ÆC07
OR LOAD
LOAD      M13518	// R_3rd STEP#08
AND       M13538	// STEP A¢Ò¡ÆC08
OR LOAD
LOAD      M13519	// R_3rd STEP#09
AND       M13539	// STEP A¢Ò¡ÆC09
OR LOAD
LOAD      M1351A	// R_3rd STEP#10
AND       M1353A	// STEP A¢Ò¡ÆC10
OR LOAD
LOAD      M1351B	// R_3rd STEP#11
AND       M1353B	// STEP A¢Ò¡ÆC11
OR LOAD
LOAD      M1351C	// R_3rd STEP#12
AND       M1353C	// STEP A¢Ò¡ÆC12
OR LOAD
LOAD      M1351D	// R_3rd STEP#13
AND       M1353D	// STEP A¢Ò¡ÆC13
OR LOAD
LOAD      M1351E	// R_3rd STEP#14
AND       M1353E	// STEP A¢Ò¡ÆC14
OR LOAD
LOAD      M1351F	// R_3rd STEP#15
AND       M1353F	// STEP A¢Ò¡ÆC15
OR LOAD
AND LOAD
AND NOT   T1080	// R_3rd MAND STEP DELAY TM
AND       M13580	// R_3rd MAND CYCLE RUN
OUT       M13500	// R_3rd AUTO TOTAL

